(* CoDeSys 2.3 project: cy-159-wg-004.pro *)
(* Title: ClevergyAS - Albino E-02 *)
(* Version: 1.25 *)
(* Author: Andrea Ravasio *)
(* Libraries: mod_com.lib 2.12.10 13:48:32, SerComm.lib 31.5.11 07:54:36, Serial_Interface_01.lib 22.4.13 11:50:14, Standard.lib 2.12.10 13:48:34, Util.lib 26.9.14 09:12:46, Modb_l05.lib 13.5.15 09:30:08, Visual.lib 2.12.10 13:48:34, Ethernet.lib 2.12.10 13:48:32, WagoLibIdent.lib 25.2.13 10:12:16, WagoLibMBX_01.lib 20.3.12 15:32:40, WagoLibStatus.lib 2.12.10 13:48:32, SysLibFile.lib 2.12.10 13:48:34, SysLibRtc.lib 2.12.10 13:48:32, SysLibSockets.lib 10.2.11 08:20:54, SysLibEvent.lib 2.12.10 13:48:34, SysLibPlcCtrl.lib 2.12.10 13:48:32, SysLibCallback.lib 2.12.10 13:48:32, WagoLibModbus_IP_01.lib 24.7.13 14:05:58, WagoLibInfo.lib 25.2.13 09:58:44 *)

(* PLC configuration (modules and I/O channels)
0750-1506 8DI / 8DO 24V DC 0.5A [Type_34_8_Channels] node 0, in %IB128 out %QB120 {INTTypePAAssignment = PLC; INTTypeModule = plugged}
  VPN_ST1 AT %IX64.0 [BOOLOnX_I] Ch_1 Digital input
  LAMP_AL AT %QX60.0 [BOOLOnX_Q] Ch_1 Digital output
  KEY_QE_ST AT %IX64.1 [BOOLOnX_I] Ch_2 Digital input
  AT %QX60.1 [BOOLOnX_Q] Ch_2 Digital output
  AT %IX64.2 [BOOLOnX_I] Ch_3 Digital input
  AT %QX60.2 [BOOLOnX_Q] Ch_3 Digital output
  AT %IX64.3 [BOOLOnX_I] Ch_4 Digital input
  AT %QX60.3 [BOOLOnX_Q] Ch_4 Digital output
  AT %IX64.4 [BOOLOnX_I] Ch_5 Digital input
  AT %QX60.4 [BOOLOnX_Q] Ch_5 Digital output
  AT %IX64.5 [BOOLOnX_I] Ch_6 Digital input
  AT %QX60.5 [BOOLOnX_Q] Ch_6 Digital output
  AT %IX64.6 [BOOLOnX_I] Ch_7 Digital input
  AT %QX60.6 [BOOLOnX_Q] Ch_7 Digital output
  AT %IX64.7 [BOOLOnX_I] Ch_8 Digital input
  AT %QX60.7 [BOOLOnX_Q] Ch_8 Digital output
0750-0652#24 RS-232/RS-485 Interface adjustable (24 Bytes) [Type_30_1_Channels] node 0, in %IB124 out %QB120 {INTTypePAAssignment = PLC; INTTypeModule = plugged}
  AT %IB0 [BYTEOnB_I] First Byte of 24
  AT %QB0 [BYTEOnB_Q] First Byte of 24
0750-0652#24 RS-232/RS-485 Interface adjustable (24 Bytes) [Type_30_1_Channels] node 0, in %IB124 out %QB120 {INTTypePAAssignment = PLC; INTTypeModule = plugged}
  AT %IB24 [BYTEOnB_I] First Byte of 24
  AT %QB24 [BYTEOnB_Q] First Byte of 24
0750-0652#24 RS-232/RS-485 Interface adjustable (24 Bytes) [Type_30_1_Channels] node 0, in %IB148 out %QB144 {INTTypePAAssignment = PLC; INTTypeModule = plugged}
  AT %IB48 [BYTEOnB_I] First Byte of 24
  AT %QB48 [BYTEOnB_Q] First Byte of 24
0750-0652#24 RS-232/RS-485 Interface adjustable (24 Bytes) [Type_30_1_Channels] node 0, in %IB172 out %QB168 {INTTypePAAssignment = PLC; INTTypeModule = plugged}
  AT %IB72 [BYTEOnB_I] First Byte of 24
  AT %QB72 [BYTEOnB_Q] First Byte of 24
0750-0652#24 RS-232/RS-485 Interface adjustable (24 Bytes) [Type_30_1_Channels] node 0, in %IB196 out %QB192 {INTTypePAAssignment = PLC; INTTypeModule = plugged}
  AT %IB96 [BYTEOnB_I] First Byte of 24
  AT %QB96 [BYTEOnB_Q] First Byte of 24
AI_PX01 AT %IW60 [WORDOnW_I] Ch_1 Input word
AI_PX02 AT %IW61 [WORDOnW_I] Ch_2 Input word
AI_PX03 AT %IW62 [WORDOnW_I] Ch_1 Input word
AI_PX04 AT %IW63 [WORDOnW_I] Ch_2 Input word
Fieldbus variables [FB_VARS] node 1, in %IB0 out %QB0
Flag variables [FLAG_VARS] node 2, in %IB0 out %QB0
Modbus-Master [MB_MASTER] node 3, in %IB0 out %QB0
*)

(* Global variable list: Global_Constants *)
VAR_GLOBAL CONSTANT

	Plant_NAME			: STRING :='cySN: 159 cyVER: Supervisione Eredi Gnutti  ';
	Plant_SN			: DWORD  :=159;	(* S/N Impianto di telecontrollo *)
	Plant_SW_VER		: WORD   :=0;	(* Versione SW installata *)


(* Configurazione Analizzatori di rete *)

	Plant_ANZ_INEPRO						: BYTE	 :=5;
	MODBUS_INEPRO_MAX_DEVICE		: BYTE:=Plant_ANZ_INEPRO;
	MODBUS_INEPRO_MAX_REG			: BYTE:=26;

	MODBUS_INEPRO_TIME_OUT			:TIME:=T#500MS;
	ANZ_INEPRO_POLLING_TIME			:TIME:=T#4S;


	(* Filesystem *)
	FilesPath  			: STRING :='S:\';

	(* TCP Logger *)
	Logger_SERVER		: STRING:='';
	Logger_IP			: STRING:='178.33.227.41'; (*'192.168.100.3';*)
	Logger_PORT			: WORD  :=80;
	Logger_GETSTART		: STRING:='GET /cygmsrv/hsgm.ashx?';
	Logger_GETEND		: STRING:='$R$N$R$N';
	Logger_CHECK		: STRING:='True';
	Logger_CRLF			: STRING:='$R$N';
	Logger_DataFile		: STRING:='S:\LOG.DAT';
	Logger_DataFileOld	: STRING:='S:\LOG.BCK';
	Logger_IndexFile	: STRING:='S:\LOG.IDX';
	Logger_ConnRetries	: BYTE:=5;
	Logger_RecoverMsgs	: BYTE:=25;

	(* TCP Remote *)
	Remote_PORT			: WORD  :=10;
	Remote_WELCOME		: STRING:='Connected$R$N';
	Remote_OK			: STRING:='OK$R$N';
	Remote_ERROR		: STRING:='ERROR$R$N';

	(* TCP Sockets *)
	MAX_SEND_TCP_SERVER					 : DWORD:=60000;(*60000*)
	MAX_RECEIVE_TCP_SERVER				 : DWORD:=3000;
	MAX_RECEIVE_TCP_SERVER_SOCKET	 	 : DWORD:=1500;
	MAX_SEND_TCP_CLIENT					 : DWORD:=15000;(*15000*)
	MAX_RECEIVE_TCP_CLIENT				 : DWORD:=1500;
	MAX_RECEIVE_TCP_CLIENT_SOCKET		 : DWORD:=1500;
	MAX_RECEIVE_UDP_SERVER				 : INT  :=1472;
	MAX_RECEIVE_UDP_CLIENT				 : INT  :=1472;
	CONNECT_WATCHDOG_TIME				 : TIME :=t#10s;


	(* VISU COLORS *)
	COLOR_RED 			: DWORD:=16#2020F0;
	COLOR_YELLOW		: DWORD:=16#20F0F0;
	COLOR_GREEN			: DWORD:=16#20F020;
	COLOR_GREEN_OFF 	: DWORD:=16#006000;
	COLOR_LBLUE			: DWORD:=16#F0F080;
	COLOR_LIGHT_GREEN	: DWORD := 16#006000;


END_VAR

(* Global variable list: Global_Retain *)
VAR_GLOBAL RETAIN PERSISTENT
	CAL01_Clima : typ_Clima;
	VRD01_Clima : typ_Clima;
	VRD02_Clima : typ_Clima;
	VRD03_Clima : typ_Clima;
	VRD04_Clima : typ_Clima;

	CTL01_Count : DWORD;

	Mode_Manual : BOOL := FALSE;


	DelayAllarmeTemperaturaNonRaggiunta: INT;
	DeltaInterventoAllarmeTempeaturaNonRaggiuta: INT;
	OffsetSetPointManuale: INT;							(* Offset al Setpoint manuale per comensare lo scambiatore *)
	OffsetSetPointManuale2: INT;						(* Offset al Setpoint manuale per comensare lo scambiatore Aggiuntivo *)
	BitAbilitaBoost: BOOL:=TRUE;						(* Abilitiazione Boost *)
	RifOffsetBoost:INT;									(* Offset al Setpoint della Caldaia per azione di Boost *)

	SogliaMinStartAntigelo: INT;
	SogliaMinStopAntigelo: INT;
	BitAbilitaAntigelo: BOOL:=TRUE;


END_VAR

(* Global variable list: Global_Variables *)
VAR_GLOBAL

	SYS    : typ_SYS;
	Logger : typ_Logger;

	Lamp	:	LAMP_AL_GENERALE;

	T_AMB	:	INT;		(* Environment temperature *)






	(* COMPRESSORI NUOVI COM 01*)
	COMPRESSORE01	:obj_COMPRESSORE_NEW := (ID:=1, Address:=1);
	COMPRESSORE05	:obj_COMPRESSORE_NEW := (ID:=5, Address:=2);

	COMPRESSORE02	:obj_COMPRESSORE_OLD := (ID:=2, Address:=1);
	COMPRESSORE03	:obj_COMPRESSORE_OLD := (ID:=3, Address:=2);
	COMPRESSORE04	:obj_COMPRESSORE_OLD := (ID:=4, Address:=3);

	ESSICATORE01	:obj_ESSICATORE_NEW := (ID:=1, Address:=1);
	ESSICATORE02	:obj_ESSICATORE := (ID:=2, Address:=2);

	FPT01:obj_MisPortata_MB:= (ID:=1, Address:=1);

	(** Communication **)
	(* ModBus TCP *)


(*	MODB06	:	obj_MODBUS_TCP 	:= (ID:=6); *)


	FPT02	:obj_MisPortata_ETH := (ID:=2, IP:='192.168.2.75');		(* misuratori di portata *)
	FPT03	:obj_MisPortata_ETH := (ID:=3, IP:='192.168.2.76');		(* misuratori di portata *)
	FPT04	:obj_MisPortata_ETH := (ID:=4, IP:='192.168.2.77');		(* misuratori di portata *)
	FPT05	:obj_MisPortata_ETH := (ID:=5, IP:='192.168.2.78');		(* misuratori di portata *)
	FPT06	:obj_MisPortata_ETH := (ID:=6, IP:='192.168.2.79');		(* misuratori di portata *)
	FPT07	:obj_MisPortata_ETH := (ID:=7, IP:='192.168.2.80');		(* misuratori di portata *)
	FPT08	:obj_MisPortata_ETH := (ID:=8, IP:='192.168.2.81');		(* misuratori di portata *)
	FPT09	:obj_MisPortata_ETH := (ID:=9, IP:='192.168.2.82');		(* misuratori di portata *)
	FPT10	:obj_MisPortata_ETH := (ID:=10, IP:='192.168.2.83');		(* misuratori di portata *)

	(* ModBus RTU  *)
(*	MODB01	:	obj_MODBUS		:= (ID:=1, COM:=2, BAUDRATE:=BAUD_19200,RS485:=TRUE,MB_timeOut:=t#500ms);   *)					 (* ANZ *)
	MODB02	:	obj_MODBUS	:= (ID:=2, COM:=3, BAUDRATE:=BAUD_9600 ,N_STOPBits:=1,RS485:=TRUE,MB_timeOut:=t#500ms);	(* COMPPRESSORI NUOVI *)
	MODB03	:	obj_MODBUS		:= (ID:=3, COM:=4, BAUDRATE:=BAUD_9600,N_STOPBits:=1,RS485:=TRUE,MB_timeOut:=t#500ms);	(* COMPRESSORI VECCHI *)
	MODB04	:	obj_MODBUS_Free		:= (ID:=4, COM:=5, BAUDRATE:=BAUD_9600,N_STOPBits:=1,RS485:=TRUE,MB_timeOut:=t#1s);  (*ESSICATORI *)
	MODB05	:	obj_MODBUS 		:= (ID:=5, COM:=6, BAUDRATE:=BAUD_9600,N_STOPBits:=1,RS485:=TRUE,MB_timeOut:=t#1s);  (*FTP01 *)





	(* Define the handler for the ModBus communication	*)
	MODB01		:	obj_MODBUS_ANZ := (ID:=1, COM:=2,
						(* TIME_OUT_TIME:= TIME_OUT_TIME:=MODBUS_INEPRO_TIME_OUT,*)
						 BAUDRATE:=BAUD_9600,
						  RS485:=TRUE,PARITY:=PARITY_EVEN,STOP_BITS:=STOPBITS_1 );


	ANZ_MODBUS_CONNECTOR_INEPRO	:	ARRAY[1..Plant_ANZ_INEPRO] OF obj_MODBUS_GENERIC_CONNECTOR;
	ANZ_INEPRO									:	ARRAY[1..Plant_ANZ_INEPRO] OF obj_ANZ_INEPRO_PRO380;

	MODBUS_INEPRO_RegDescr 				: ARRAY[1..MODBUS_INEPRO_MAX_DEVICE, 1..MODBUS_INEPRO_MAX_REG] OF STRING(20);
	MODBUS_INEPRO_RegAddress			 : ARRAY[1..MODBUS_INEPRO_MAX_DEVICE, 1..MODBUS_INEPRO_MAX_REG] OF WORD;
	MODBUS_INEPRO_RegQuantity 			: ARRAY[1..MODBUS_INEPRO_MAX_DEVICE, 1..MODBUS_INEPRO_MAX_REG] OF BYTE;
	MODBUS_INEPRO_RegValueType			 : ARRAY[1..MODBUS_INEPRO_MAX_DEVICE, 1..MODBUS_INEPRO_MAX_REG] OF en_Modbus_Reg_Type;




(* CONFIGURAZIONE INGRESSI ANALOGICI 4-20mA  *)

	PX01  : obj_AI_GEN	:= ( ID:=1 ,
								SogliaHL:=4096 ,   	 	(* Soglia Sonda Aperta = 2,5mA *)
								SogliaHH:=32767,	 	(* Soglia Sonda CC = 20mA *)
								SogliaWL:=10, 			(* Soglia WRN Bassa  *)
								SogliaWH:=140,			(* Soglia WRN Alta   *)
								PuntoMinX:=0, 		   	 (* Scalatura Minima vedi data di targa sonda 0 bar *)
								PuntoMaxX:=160,			(* Scalatura Massima Vedi data di targa Sonda 16.0bar *)
								PuntoMinY:=6553,			(* Valore minimio per scalatura = 4mA *)
								PuntoMaxY:=32767,		(* Valore Massimo per Scalatura = 20mA *)
								Decimali:=0,				(* Decimali da ottenere durante la scalatura *)
								TipoSensore:='PPV'		(* Riferimento nle file LOG *)
								);

	PX02  : obj_AI_GEN	:= ( ID:=2 ,
								SogliaHL:=4096 ,   	 	(* Soglia Sonda Aperta = 2,5mA *)
								SogliaHH:=32767,	 	(* Soglia Sonda CC = 20mA *)
								SogliaWL:=10, 			(* Soglia WRN Bassa *)
								SogliaWH:=120,			(* Soglia WRN Alta *)
								PuntoMinX:=0, 		   	 (* Scalatura Minima vedi data di targa sonda  0 bar*)
								PuntoMaxX:=160,			(* Scalatura Massima Vedi data di targa Sonda 16.0bar  *)
								PuntoMinY:=6553,			(* Valore minimio per scalatura = 4mA *)
								PuntoMaxY:=32767,		(* Valore Massimo per Scalatura = 20mA *)
								Decimali:=0,				(* Decimali da ottenere durante la scalatura *)
								TipoSensore:='PPV'		(* Riferimento nle file LOG *)
								);

	PX03  : obj_AI_GEN	:= ( ID:=3 ,
								SogliaHL:=4096 ,   	 	(* Soglia Sonda Aperta = 2,5mA *)
								SogliaHH:=32767,	 	(* Soglia Sonda CC = 20mA *)
								SogliaWL:=10, 			(* Soglia WRN Bassa  = *)
								SogliaWH:=120,			(* Soglia WRN Alta  =  *)
								PuntoMinX:=0, 		   	 (* Scalatura Minima vedi data di targa sonda  0 bar*)
								PuntoMaxX:=160,			(* Scalatura Massima Vedi data di targa Sonda 16.0bar *)
								PuntoMinY:=6553,			(* Valore minimio per scalatura = 4mA *)
								PuntoMaxY:=32767,		(* Valore Massimo per Scalatura = 20mA *)
								Decimali:=0,				(* Decimali da ottenere durante la scalatura *)
								TipoSensore:='PPV'		(* Riferimento nle file LOG *)
								);

	PX04  : obj_AI_GEN	:= ( ID:=4 ,
								SogliaHL:=4096 ,   	 	(* Soglia Sonda Aperta = 2,5mA *)
								SogliaHH:=32767,	 	(* Soglia Sonda CC = 20mA *)
								SogliaWL:=10, 			(* Soglia WRN Bassa  =  *)
								SogliaWH:=120,			(* Soglia WRN Alta  =  *)
								PuntoMinX:=0, 		   	 (* Scalatura Minima vedi data di targa sonda 0 bar *)
								PuntoMaxX:=160,			(* Scalatura Massima Vedi data di targa Sonda 16.0bar *)
								PuntoMinY:=6553,			(* Valore minimio per scalatura = 4mA *)
								PuntoMaxY:=32767,		(* Valore Massimo per Scalatura = 20mA *)
								Decimali:=0,				(* Decimali da ottenere durante la scalatura *)
								TipoSensore:='PPV'		(* Riferimento nle file LOG *)
								);





(* interblocchi comunicazione modbus *)

	NodoDaInterrogareCompressoreNuovo: BYTE;
	InibiscoModbusCompressoreNuovo: BOOL;

	NodoDaInterrogareCompressoreVecchio: BYTE;
	InibiscoModbusCompressoreVecchio: BOOL;

	NodoDaInterrogareMisuratoreDiPortata: BYTE;
	InibiscoModbusMisuratoreDiPortata: BOOL;

	NodoDaInterrogareMisuratoreDiPortata_ETH: BYTE;

	NodoDaInterrogareEssicatore: BYTE;
	InibiscoModbusEssicatore: BOOL;



END_VAR

(* Data type in LON/Enumerations *)
TYPE alarm_type_t :
(
	AL_HEADER := -13,
	AL_FOOTER := -12,
	AL_DEBUG := -11,
	AL_INFO := -10,
	AL_SYSTEM_INFO := -6,
	AL_VALUE_INVALID := -5,
	AL_CONSTANT := -4,
	AL_OFFLINE := -3,
	AL_UNKNOWN := -2,
	AL_NUL := -1,
	AL_NO_CONDITION := 0,
	AL_ALM_CONDITION := 1,
	AL_TOT_SVC_ALM_1 := 2,
	AL_TOT_SVC_ALM_2 := 3,
	AL_TOT_SVC_ALM_3 := 4,
	AL_LOW_LMT_CLR_1 := 5,
	AL_LOW_LMT_CLR_2 := 6,
	AL_HIGH_LMT_CLR_1 := 7,
	AL_HIGH_LMT_CLR_2 := 8,
	AL_LOW_LMT_ALM_1 := 9,
	AL_LOW_LMT_ALM_2 := 10,
	AL_HIGH_LMT_ALM_1 := 11,
	AL_HIGH_LMT_ALM_2 := 12,
	AL_FIR_ALM := 13,
	AL_FIR_PRE_ALM := 14,
	AL_FIR_TRBL := 15,
	AL_FIR_SUPV := 16,
	AL_FIR_TEST_ALM := 17,
	AL_FIR_TEST_PRE_ALM := 18,
	AL_FIR_ENVCOMP_MAX := 19,
	AL_FIR_MONITOR_COND := 20,
	AL_FIR_MAINT_ALERT := 21,
	AL_FATAL_ERROR := 30,
	AL_ERROR := 31,
	AL_WARNING := 32
);
END_TYPE

(* Data type in DT_ANZ *)
TYPE en_ANZ_Type :
(
	THREE_PHASE			:=0,
	MONO_PHASE			:=1
);
END_TYPE

(* Data type in Errors *)
TYPE en_Logger_ErrLev :
(
	EL_Log			:=0,
	EL_Wrn			:=1,
	EL_Alarm		:=2,
	EL_AlarmStop	:=3
);
END_TYPE

(* Data type in Errors *)
TYPE en_Logger_Status :
(
	S_Logger_UNKNOWN := 0,
	S_Logger_IDLE,
	S_Logger_WAITCONN,
	S_Logger_WAITTX,
	S_Logger_WAITRESP,
	S_Logger_ERROR
);
END_TYPE

(* Data type *)
TYPE en_Modbus_Reg_Type :
(
	VALUE_REAL		:=0,
	VALUE_LONG		:=4
);
END_TYPE

(* Data type *)
TYPE en_SYS_Objects :
(
	EO_SYS		:=0,  (* PLC *)
	EO_VPN		:=1,  (* VPN *)
	EO_DOOR		:=2,  (* Door & access control *)

	EO_CAL		:=10, (* Caldaia *)
	EO_CIR		:=11, (* Circolatore *)
	EO_CRON		:=12, (* Crono-termostato *)
	EO_VRD		:=13, (* Valvola miscelatore pannelli *)
	EO_CTL		:=14, (* Contalitri *)
	EO_CTB		:=15, (* Contabilizzatore *)
	EO_TPV		:=16, (* Temperature probes values *)
	EO_PPV		:=17, (* Pressure probes values *)
	EO_PBV		:=18, (* Over-Pressure Alarms *)
	EO_TBV		:=19, (* Over-Temperature Alarms *)
	EO_PMV		:=20, (* Under-Pressure Alarms *)
	EO_GRU		:=21, (* Gruppo termico *)
	EO_PDC		:=22, (* Pompa di calore *)
	EO_SOL		:=23, (* Pannello solare termico *)
	EO_ESOL		:=24, (* Pannello solare fotovoltaico *)
	EO_GAS		:=25, (* Contatore GAS *)
	EO_PORT		:=26, (* Misuratore di portata *)
	EO_FPV		:=27, (* Flow probes values *)
	EO_ANZ		:=28, (* Analizzatore di rete *)
	EO_SCA		:=29, (* Signal Control Alarms *)
	EO_LUX		:=30, (* Base Illumination point *)
	EO_LUXM		:=31, (* Metered Illumination point *)
	EO_PSG		:=32, (* Sensore di passaggio *)
	EO_HVAC		:=33, (* Heating, Ventilating and Air Conditioning *)
	EO_HYGRV	:=34, (* Relative Humidity sensors value *)
	EO_COOV		:=35, (* Carbon Dioxide CO2 sensors value *)
	EO_INV		:=36, (* Inverter *)
	EO_STR		:=37, (* Smart string box *)

	EO_CIRD		:=39, (* Double CIR *)
	EO_ACS		:=40, (* Hot domestic water *)
	EO_FRG		:=41, (* Frigo *)
	EO_THER		:=42, (* Thermostat *)
	EO_CIRM		:=43, (* Modbus CIR *)
	EO_CIRDM	:=44, (* Modbus double CIR *)
	EO_UTA		:=47, (* Modbus double CIR *)

	EO_FPT		:=53, (* Flow Pressure Temperature	FPTxx *)


	EO_ZGW			:=200,  (* ZigBee - Gateway *)
	EO_ZRM			:=201,	(* ZigBee - Repeater *)
	EO_ZREL			:=202,	(* ZigBee - Actuator rele *)
	EO_ZTHL			:=203,	(* ZigBee - Temperature Sensor *)

	EO_ASGW			:=250,	(* ASi - Gateway *)
	EO_ASCBI		:=251,	(* ASi - Input Board, Ciabatta *)

	EO_LON			:=1000, (* Bus - LON *)
	EO_MODBUS		:=1001, (* Bus - MODBUS *)
	EO_MBUS			:=1002, (* Bus - M-BUS *)
	EO_MODBUS_TCP	:=1003, (* Bus - MODBUS TCP *)




	EO_COMPINGRR		:=10000,		(*Compressore Ingerson Rand R225 NE *)
	EO_COMPINGRML	:=	10001,		(*Compressore Ingerson Rand ML250SSR *)
	EO_ESC				:=	10002,		(*Essicatore *)





	EO_GENERIC		:=9000, (* Generic dataset *)
	EO_EXPO			:=9001 (* EXPO dataset *)
);
END_TYPE

(* Data type *)
TYPE en_SYS_Status :
(
	S_UNKNOWN  := 0,
	S_STARTUP,
	S_INIT_RTC,
	S_INIT_VAR,
	S_AUTOTEST,
	S_RUNNING,
	S_SHUTDOWN,
	S_HALT
);
END_TYPE

(* Data type in LON/Enumerations *)
TYPE file_request_t :
(
	FR_NUL := -1,
	FR_OPEN_TO_SEND := 0,
	FR_OPEN_TO_RECEIVE := 1,
	FR_CLOSE_FILE := 2,
	FR_CLOSE_DELETE_FILE := 3,
	FR_DIRECTORY_LOOKUP := 4,
	FR_OPEN_TO_SEND_RA := 5,
	FR_OPEN_TO_RECEIVE_RA := 6
);
END_TYPE

(* Data type in LON/Enumerations *)
TYPE file_status_t :
(
	FS_NUL := -1,
	FS_XFER_OK := 0,
	FS_LOOKUP_OK := 1,
	FS_OPEN_FAIL := 2,
	FS_LOOKUP_ERR := 3,
	FS_XFER_UNDERWAY := 4,
	FS_IO_ERR := 5,
	FS_TIMEOUT_ERR := 6,
	FS_WINDOW_ERR := 7,
	FS_AUTH_ERR := 8,
	FS_ACCESS_UNAVAIL := 9,
	FS_SEEK_INVALID := 10,
	FS_SEEK_WAIT := 11
);
END_TYPE

(* Data type in LON/Enumerations *)
TYPE hvac_t :
(
	HVAC_NUL := -1,
	HVAC_AUTO := 0,
	HVAC_HEAT := 1,
	HVAC_MRNG_WRMUP := 2,
	HVAC_COOL := 3,
	HVAC_NIGHT_PURGE := 4,
	HVAC_PRE_COOL := 5,
	HVAC_OFF := 6,
	HVAC_TEST := 7,
	HVAC_EMERG_HEAT := 8,
	HVAC_FAN_ONLY := 9,
	HVAC_FREE_COOL := 10,
	HVAC_ICE := 11,
	HVAC_MAX_HEAT := 12,
	HVAC_ECONOMY := 13,
	HVAC_DEHUMID := 14,
	HVAC_CALIBRATE := 15,
	HVAC_EMERG_COOL := 16,
	HVAC_EMERG_STEAM := 17,
	HVAC_MAX_COOL := 18,
	HVAC_HVC_LOAD := 19,
	HVAC_NO_LOAD := 20
);
END_TYPE

(* Data type in LON/Enumerations *)
TYPE object_request_t :
(
	RQ_NUL := -1,
	RQ_NORMAL := 0,
	RQ_DISABLED := 1,
	RQ_UPDATE_STATUS := 2,
	RQ_SELF_TEST := 3,
	RQ_UPDATE_ALARM := 4,
	RQ_REPORT_MASK := 5,
	RQ_OVERRIDE := 6,
	RQ_ENABLE := 7,
	RQ_RMV_OVERRIDE := 8,
	RQ_CLEAR_STATUS := 9,
	RQ_CLEAR_ALARM := 10,
	RQ_ALARM_NOTIFY_ENABLED := 11,
	RQ_ALARM_NOTIFY_DISABLED := 12,
	RQ_MANUAL_CTRL := 13,
	RQ_REMOTE_CTRL := 14,
	RQ_PROGRAM := 15,
	RQ_CLEAR_RESET := 16,
	RQ_RESET := 17,
	RQ_CLEAR_LOG := 18,
	RQ_LOAD_PROGRAM := 19,
	RQ_RUN_PROGRAM := 20,
	RQ_HALT_PROGRAM := 21,
	RQ_RESTART_PROGRAM := 22,
	RQ_UNLOAD_PROGRAM := 23,
	RQ_STEP_PROGRAM := 24
);
END_TYPE

(* Data type in LON/Enumerations *)
TYPE priority_level_t :
(
	PR_NUL := -1,
	PR_LEVEL_0 := 0,
	PR_LEVEL_1 := 1,
	PR_LEVEL_2 := 2,
	PR_LEVEL_3 := 3,
	PR_1 := 4,
	PR_2 := 5,
	PR_3 := 6,
	PR_4 := 7,
	PR_6 := 8,
	PR_8 := 9,
	PR_10 := 10,
	PR_16 := 11
);
END_TYPE

(* Data type in DT_ANZ *)
(*
	typ_ANZ_3P 

	Data that each ANZ 3-phase block must provide (to the Clevergy platform).
*)
TYPE typ_ANZ :
STRUCT

	(* voltages *)
	V_L1N		:	DWORD;	(* V *)
	V_L2N		:	DWORD;
	V_L3N		:	DWORD;
	V_L1L2		:	DWORD;
	V_L2L3		:	DWORD;
	V_L3L1		:	DWORD;

	(* frequency *)
	FREQ		:	DWORD;	(* E-3 Hz *) (* rif. L1 *)

	(* currents *)
	I_L1			:	DWORD;	(* E-3 A *)
	I_L2			:	DWORD;
	I_L3			:	DWORD;
	I_L1_Max		:	DWORD;	(* E-3 A *)
	I_L2_Max		:	DWORD;
	I_L3_Max		:	DWORD;

	(* power factors *)
	PF_L1		:	DINT;	(* E-3 *)
	PF_L2		:	DINT;
	PF_L3		:	DINT;

	(* active powers *)
	P_3P			:	DINT;   (* W *)
	P_3P_Avg		:	DINT;
	P_3P_Max	:	DINT:=0;

	(* reactive powers *)
	Q_3P		:	DINT;	(* VAr *)
	Q_3P_Max	:	DINT:=-2147483648;	(* VAr *)

	(* active energy *)
	WH_3P		:	DWORD;	(* Wh *)

	(* reactive energy *)
	VARH_3P		:	DINT;	(* VArh *)

	(* cosphi *)
	COSPHI_L1		:	DINT;	(* E-3 *)
	COSPHI_L2		:	DINT;	(* E-3 *)
	COSPHI_L3		:	DINT;	(* E-3 *)

END_STRUCT
END_TYPE

(* Data type in DT_ANZ_INEPRO_PRO380 *)
TYPE typ_ANZ_INEPRO_PRO380 :
STRUCT

		rTotalActivePower					: REAL;
		rTotalReactivePower				: REAL;
		rTotalApparentPower				: REAL;
		rTotalPowerFactorPF				: REAL;
		rTotalActiveEnergy					: REAL;
		rTotalReactiveEnergy				: REAL;

		arCurrent							: ARRAY[1..3] OF REAL;
		arVoltage_L_N						: ARRAY[1..3] OF REAL;
		arActivePower						: ARRAY[1..3] OF REAL;
		arReactivePower					: ARRAY[1..3] OF REAL;
		arApparentPower					: ARRAY[1..3] OF REAL;

		arPowerFactorPF					: ARRAY[1..3] OF REAL;
		arFrequency						:REAL;


		rMaximumCurrentL1			: REAL;
		rMaximumCurrentL2				: REAL;
		rMaximumCurrentL3			: REAL;


		rMaximumTotalActivePower			: REAL :=0;
		rAverageTotalActivePower 			: REAL :=0;

		rMaximumTotalReactivePower		: REAL :=0;

END_STRUCT
END_TYPE

(* Data type in DT_ANZ *)
(*
	typ_ANZ_3P 

	Data that each ANZ 3-phase block must provide (to the Clevergy platform).
*)
TYPE typ_ANZ_REAL :
STRUCT

	(* voltages *)
	V_L1N		:	REAL;	(* V *)
	V_L2N		:	REAL;
	V_L3N		:	REAL;
	V_L1L2		:	REAL;
	V_L2L3		:	REAL;
	V_L3L1		:	REAL;

	(* frequency *)
	FREQ		:	REAL;	(* E-3 Hz *) (* rif. L1 *)

	(* currents *)
	I_L1			:	REAL;	(* E-3 A *)
	I_L2			:	REAL;
	I_L3			:	REAL;
	I_L1_Max		:	REAL;	(* E-3 A *)
	I_L2_Max		:	REAL;
	I_L3_Max		:	REAL;

	(* power factors *)
	PF_L1		:	REAL;	(* E-3 *)
	PF_L2		:	REAL;
	PF_L3		:	REAL;

	(* active powers *)
	P_3P			:	REAL;   (* W *)
	P_3P_Avg		:	REAL;
	P_3P_Max	:	REAL:=0;

	(* reactive powers *)
	Q_3P		:	REAL;	(* VAr *)
	Q_3P_Max	:	REAL:=-2147483648;	(* VAr *)

	(* active energy *)
	WH_3P		:	REAL;	(* Wh *)

	(* reactive energy *)
	VARH_3P		:	REAL;	(* VArh *)

	(* cosphi *)
	COSPHI_L1		:	REAL;	(* E-3 *)
	COSPHI_L2		:	REAL;	(* E-3 *)
	COSPHI_L3		:	REAL;	(* E-3 *)

END_STRUCT
END_TYPE

(* Data type in Plant_Objects *)
TYPE typ_Clima : (* CURVA CLIMATICA *)
STRUCT
	InitOK:		BOOL;
	Points: 	ARRAY [0..10] OF POINT;
END_STRUCT
END_TYPE

(* Data type in Plant_Objects *)
TYPE typ_Cron_Calendar :
STRUCT
	Profile		: ARRAY[0..384] OF BYTE;
END_STRUCT
END_TYPE

(* Data type in Plant_Objects *)
TYPE typ_Cron_Jolly :
STRUCT
	Start		: DT;
	End			: DT;
	Temp		: WORD;
	Flags		: WORD; (* B0:Enabled B1..B15:Unused *)
END_STRUCT
END_TYPE

(* Data type in Plant_Objects *)
TYPE typ_Cron_Profile :
STRUCT
	Flags		: WORD;
	Setpoint	: ARRAY [0..95] OF WORD;
END_STRUCT
END_TYPE

(* Data type in Errors *)
TYPE typ_Logger :
STRUCT
	Status		: en_Logger_Status;

	SendReq		: BOOL;
	SendIdx		: DWORD;
	SendData	: ARRAY [0..MAX_SEND_TCP_CLIENT] OF BYTE;
	SendLen		: DINT;

	TData		: ARRAY [0..MAX_SEND_TCP_CLIENT] OF BYTE;
	TLen		: DINT;

	LastIdxPos	: DWORD;

	(* Temporary variables used by objects *)
	s1			: STRING(256);
	i1			: WORD;


END_STRUCT
END_TYPE

(* Data type in Plant_Objects *)
TYPE typ_MODBUS_VAR : (* Gestione parametri MODBUS *)
STRUCT
	SlaveAddress	: BYTE;
	FunCode			: BYTE;
	FunAddress		: WORD;
	Refresh_Time	: BYTE; (* 0:No refresh x:Refresh in seconds *)
	Refresh_Cnt		: BYTE; (* INTERNAL *)
	Variable		: POINTER TO WORD;
	Variable_Size	: BYTE;
	Variable_Mirror : WORD; (* INTERNAL [Force refresh on read variables when <>0] *)
END_STRUCT
END_TYPE

(* Data type in Plant_Objects *)
TYPE typ_MODBUS_VAR_ANZ : (* Gestione parametri MODBUS *)
STRUCT
	SlaveAddress	: BYTE;
	FunCode			: BYTE;
	FunAddress		: WORD;
	Refresh_Time	: BYTE; (* 0:No refresh x:Refresh in seconds *)
	Refresh_Cnt		: BYTE; (* INTERNAL *)
	Variable		: POINTER TO ARRAY [0..124] OF WORD;	(* For classical ModBus it has to be equal to "typModbusResponse.Data"
																that is an array of 125 word ([0..124]) *)
	Variable_Size	: BYTE;
	Variable_Mirror : WORD; (* INTERNAL [Force refresh on read variables when <>0] *)
END_STRUCT
END_TYPE

(* Data type *)
TYPE typ_SYS :
STRUCT
	Status			: en_SYS_Status;
	Warning			: BOOL;
	Alarm			: BOOL;
	AlarmStop		: BOOL;

	Time_LogString	: STRING;
	Time_Year		: WORD;
	Time_Month		: BYTE;
	Time_Day		: BYTE;

	Time_CT_DT		: DT;
	Time_CT_Day		: WORD;
	Time_CT_Quarter	: BYTE;

	LastLogs_Idx	: BYTE;
	LastLogs_Dat	: ARRAY[0..5] OF STRING;
	LastLogs_Msg	: ARRAY[0..5] OF STRING;

END_STRUCT
END_TYPE

(* Data type in LON/NetworkVariables *)
TYPE typSnvtAlarm : 
STRUCT
	abLocation : ARRAY[0..5] OF BYTE;
	wObjectId : WORD;
	bAlarmType : BYTE (* enum type alarm_type_t *);
	bPriorityLevel : BYTE (* enum type priority_level_t *);
	wIndexToSnvt : WORD;
	abValue : ARRAY[0..3] OF BYTE;
	wYear : WORD;
	bMonth : BYTE;
	bDay : BYTE;
	bHour : BYTE;
	bMinute : BYTE;
	bSecond : BYTE;
	wMillisecond : WORD;
	abAlarmLimit : ARRAY[0..3] OF BYTE;
	bStatusInformation : BYTE; (* bit allocation of bStatusInformation:
	bit 0: NVI update counter LSB
	bit 1: NVI update counter
	bit 2: NVI update counter
	bit 3: NVI update counter MSB
	bit 4: timeout for NVI occurs (MaxRcvTime expired)
	bit 5: reserved
	bit 6: reserved
	bit 7: force NVO update *)
	bInternalUseOnly : BYTE; (* Do not use this byte in your application! *)
END_STRUCT
END_TYPE

(* Data type in LON/NetworkVariables *)
TYPE typSnvtFilePos : 
STRUCT
	diRwPtr : DINT;
	wRwLength : WORD;
	bStatusInformation : BYTE; (* bit allocation of bStatusInformation:
	bit 0: NVI update counter LSB
	bit 1: NVI update counter
	bit 2: NVI update counter
	bit 3: NVI update counter MSB
	bit 4: timeout for NVI occurs (MaxRcvTime expired)
	bit 5: reserved
	bit 6: reserved
	bit 7: force NVO update *)
	bInternalUseOnly : BYTE; (* Do not use this byte in your application! *)
END_STRUCT
END_TYPE

(* Data type in LON/NetworkVariables *)
TYPE typSnvtFileReq : 
STRUCT
	bRequest : BYTE (* enum type file_request_t *);
	wIndex : WORD;
	wReceiveTimeout : WORD;
	abDestAddress : ARRAY[0..4] OF BYTE (* union declaration *);
	bAuthOn : BYTE;
	bPrioOn : BYTE;
	bStatusInformation : BYTE; (* bit allocation of bStatusInformation:
	bit 0: NVI update counter LSB
	bit 1: NVI update counter
	bit 2: NVI update counter
	bit 3: NVI update counter MSB
	bit 4: timeout for NVI occurs (MaxRcvTime expired)
	bit 5: reserved
	bit 6: reserved
	bit 7: force NVO update *)
	bInternalUseOnly : BYTE; (* Do not use this byte in your application! *)
END_STRUCT
END_TYPE

(* Data type in LON/NetworkVariables *)
TYPE typSnvtFileStatus : 
STRUCT
	bStatus : BYTE (* enum type file_status_t *);
	wNumberOfFiles : WORD;
	wSelectedFile : WORD;
	abAdr : ARRAY[0..21] OF BYTE (* union declaration *);
	bStatusInformation : BYTE; (* bit allocation of bStatusInformation:
	bit 0: NVI update counter LSB
	bit 1: NVI update counter
	bit 2: NVI update counter
	bit 3: NVI update counter MSB
	bit 4: timeout for NVI occurs (MaxRcvTime expired)
	bit 5: reserved
	bit 6: reserved
	bit 7: force NVO update *)
	bInternalUseOnly : BYTE; (* Do not use this byte in your application! *)
END_STRUCT
END_TYPE

(* Data type in LON/NetworkVariables *)
TYPE typSnvtHvacMode : 
STRUCT
	bSnvtHvacMode : BYTE (* enum type hvac_t *);
	bStatusInformation : BYTE; (* bit allocation of bStatusInformation:
	bit 0: NVI update counter LSB
	bit 1: NVI update counter
	bit 2: NVI update counter
	bit 3: NVI update counter MSB
	bit 4: timeout for NVI occurs (MaxRcvTime expired)
	bit 5: reserved
	bit 6: reserved
	bit 7: force NVO update *)
	bInternalUseOnly : BYTE; (* Do not use this byte in your application! *)
END_STRUCT
END_TYPE

(* Data type in LON/NetworkVariables *)
TYPE typSnvtObjRequest : 
STRUCT
	wObjectId : WORD;
	bObjectRequest : BYTE (* enum type object_request_t *);
	bStatusInformation : BYTE; (* bit allocation of bStatusInformation:
	bit 0: NVI update counter LSB
	bit 1: NVI update counter
	bit 2: NVI update counter
	bit 3: NVI update counter MSB
	bit 4: timeout for NVI occurs (MaxRcvTime expired)
	bit 5: reserved
	bit 6: reserved
	bit 7: force NVO update *)
	bInternalUseOnly : BYTE; (* Do not use this byte in your application! *)
END_STRUCT
END_TYPE

(* Data type in LON/NetworkVariables *)
TYPE typSnvtObjStatus : 
STRUCT
	wObjectId : WORD;
	bBitfieldByteOffset2 : BYTE (* bit field *);
	bBitfieldByteOffset3 : BYTE (* bit field *);
	bBitfieldByteOffset4 : BYTE (* bit field *);
	bBitfieldByteOffset5 : BYTE (* bit field *);
	bStatusInformation : BYTE; (* bit allocation of bStatusInformation:
	bit 0: NVI update counter LSB
	bit 1: NVI update counter
	bit 2: NVI update counter
	bit 3: NVI update counter MSB
	bit 4: timeout for NVI occurs (MaxRcvTime expired)
	bit 5: reserved
	bit 6: reserved
	bit 7: force NVO update *)
	bInternalUseOnly : BYTE; (* Do not use this byte in your application! *)
END_STRUCT
END_TYPE

(* Data type in LON/NetworkVariables *)
TYPE typSnvtState : 
STRUCT
	bBitfieldByteOffset0 : BYTE (* bit field *);
	bBitfieldByteOffset1 : BYTE (* bit field *);
	bStatusInformation : BYTE; (* bit allocation of bStatusInformation:
	bit 0: NVI update counter LSB
	bit 1: NVI update counter
	bit 2: NVI update counter
	bit 3: NVI update counter MSB
	bit 4: timeout for NVI occurs (MaxRcvTime expired)
	bit 5: reserved
	bit 6: reserved
	bit 7: force NVO update *)
	bInternalUseOnly : BYTE; (* Do not use this byte in your application! *)
END_STRUCT
END_TYPE

(* Data type in LON/NetworkVariables *)
TYPE typSnvtSwitch : 
STRUCT
	bValue : BYTE;
	siState : SINT;
	bStatusInformation : BYTE; (* bit allocation of bStatusInformation:
	bit 0: NVI update counter LSB
	bit 1: NVI update counter
	bit 2: NVI update counter
	bit 3: NVI update counter MSB
	bit 4: timeout for NVI occurs (MaxRcvTime expired)
	bit 5: reserved
	bit 6: reserved
	bit 7: force NVO update *)
	bInternalUseOnly : BYTE; (* Do not use this byte in your application! *)
END_STRUCT
END_TYPE

(* Data type in LON/NetworkVariables *)
TYPE typSnvtTempP :
STRUCT
	iSnvtTempP : INT;
	bStatusInformation : BYTE; (* bit allocation of bStatusInformation:
	bit 0: NVI update counter LSB
	bit 1: NVI update counter
	bit 2: NVI update counter
	bit 3: NVI update counter MSB
	bit 4: timeout for NVI occurs (MaxRcvTime expired)
	bit 5: reserved
	bit 6: reserved
	bit 7: force NVO update *)
	bInternalUseOnly : BYTE; (* Do not use this byte in your application! *)
END_STRUCT
END_TYPE

(* Data type in LON/NetworkVariables *)
TYPE typSnvtTimeStamp : 
STRUCT
	iYear : INT;
	bMonth : BYTE;
	bDay : BYTE;
	bHour : BYTE;
	bMinute : BYTE;
	bSecond : BYTE;
	bStatusInformation : BYTE; (* bit allocation of bStatusInformation:
	bit 0: NVI update counter LSB
	bit 1: NVI update counter
	bit 2: NVI update counter
	bit 3: NVI update counter MSB
	bit 4: timeout for NVI occurs (MaxRcvTime expired)
	bit 5: reserved
	bit 6: reserved
	bit 7: force NVO update *)
	bInternalUseOnly : BYTE; (* Do not use this byte in your application! *)
END_STRUCT
END_TYPE

(* POU PLC_PRG, ST *)
PROGRAM PLC_PRG
VAR
	Timer1: TON; (* Fast controls tick *)
	Timer2: TON; (* Plant control tick *)
	Timer3: TON; (* Logger timer *)


	status : BYTE;
	i	  : BYTE;



	HMI_AggiornaLog: BOOL;

	TempoCilcoETH: TON;
	StepETH: INT;


	Timer4: TON;
	IndiceArraRet: INT;
	pippo: BOOL;
	k: INT;
	CreaFile: obj_CreaFile;
	arra: BOOL;
	ArrayDaSalvare: ARRAY [1..80,0..60] OF STRING(10);
	record: INT;
	x: INT;


	EseguiLog: INT;
	Ton_pausaTrig: TON;
	R_TrigAggiornaLog: R_TRIG;


	TempoLog: TIME := t#500ms;
END_VAR

VAR RETAIN

END_VAR


VAR_INPUT
	RichiestaDaRemoto:BOOL;

END_VAR
(******************************************************************************
 ****                           MAIN TASK CODE                             ****
 ******************************************************************************

	Network setup:
		IP  = 192.168.2.73 | MSK = 255.255.255.0
		GW	= 192.168.2.254 | DNS = 192.168.100.1
		SNTP = 193.204.114.232 (3600s) ==> 192.168.100.3
*)





(*==============================*)
(*===== Main status machine ====*)
(*==============================*)


Main_Stm();

(*==============================*)
(*== Running cycle operations ==*)
(*==============================*)

IF SYS.Status>S_INIT_VAR THEN




	(* ModBus *)
	MODB02();

	COMPRESSORE01(ModBus:=MODB02);
	COMPRESSORE05(ModBus:=MODB02);

	NodoDaInterrogareCompressoreNuovo:=LIMIT(1,NodoDaInterrogareCompressoreNuovo,3);
	IF NodoDaInterrogareCompressoreNuovo>2 THEN NodoDaInterrogareCompressoreNuovo:=1;END_IF;


	(* ModBus *)
	MODB03();

	COMPRESSORE02(ModBus:=MODB03);
	COMPRESSORE03(ModBus:=MODB03);
	COMPRESSORE04(ModBus:=MODB03);

	NodoDaInterrogareCompressoreVecchio:=LIMIT(1,NodoDaInterrogareCompressoreVecchio,4);
	IF NodoDaInterrogareCompressoreVecchio>3 THEN NodoDaInterrogareCompressoreVecchio:=1;END_IF;


	(* ModBus *)
	MODB04();


(*	ESSICATORE01(ModBus:=MODB04); *)
	ESSICATORE02(ModBus:=MODB04);

	NodoDaInterrogareEssicatore:=LIMIT(1,NodoDaInterrogareEssicatore,3);
	IF NodoDaInterrogareEssicatore>2 THEN NodoDaInterrogareEssicatore:=2;END_IF;  (**** ma modificare nel caso si inserisca anche il nodo 1 ***)





	(* ModBus *)
	MODB05();

	FPT01(ModBus:=MODB05);

	NodoDaInterrogareMisuratoreDiPortata:=LIMIT(1,NodoDaInterrogareMisuratoreDiPortata,2);
	IF NodoDaInterrogareMisuratoreDiPortata>1 THEN NodoDaInterrogareMisuratoreDiPortata:=1;END_IF;





	TempoCilcoETH(IN:= NOT TempoCilcoETH.Q , PT:=t#1s , Q=> , ET=> );
	IF TempoCilcoETH.Q THEN StepETH:=StepETH+1;END_IF


 	FPT02();
	FPT03();
	FPT04();
	FPT05();
	FPT06();
	FPT07();
	FPT08();
	FPT09();
	FPT10();



	(*MODB06(); *)

	(* FPT02(startCom:=StepETH=2,MODBUS:=MODB06); *)
	(* FPT03(startCom:=StepETH=3  ,MODBUS:=MODB06);
	 FPT04(startCom:=StepETH=4 ,MODBUS:=MODB06);
	 FPT05(startCom:=StepETH=5 ,MODBUS:=MODB06);
	 FPT06(startCom:=StepETH=6 ,MODBUS:=MODB06);
	 FPT07(startCom:=StepETH=7 ,MODBUS:=MODB06);
	 FPT08(startCom:=StepETH=8 ,MODBUS:=MODB06);
	 FPT09(startCom:=StepETH=9 ,MODBUS:=MODB06);
	 FPT10(startCom:=StepETH=10 ,MODBUS:=MODB06); *)

	(*IF StepETH>10 THEN StepETH:=1;END_IF;
	IF NodoDaInterrogareMisuratoreDiPortata_ETH>10 THEN NodoDaInterrogareMisuratoreDiPortata_ETH:=2;END_IF; *)



END_IF


(*==============================*)
(*== System cycle operations ===*)
(*==============================*)
(* Execute TCP processes *)
Logger_Proc();
Remote_Proc();
(*
(* Update user led *)
USRLED_Update();
(* Execute Cron Editor commands *)
*)
END_PROGRAM
ACTION Main_Stm:
CASE Sys.Status OF

	S_STARTUP:
		Sys.Status:=S_INIT_RTC;

	S_INIT_RTC:
		(* Check RTC and update from network *)
		RTC_Update();
		(* Check time *)
		IF Sys.Time_Year>2000 THEN
			Sys.Status:=S_INIT_VAR;
		END_IF








	S_INIT_VAR:
		LogEv(EL_Wrn,EO_SYS,0,1,CONCAT('System_startup_v',WORD_TO_STRING(Plant_SW_VER)));
		Sys.Status:=S_RUNNING;

		OBJ_Definition();


	S_RUNNING:
		Timer1(IN:=NOT Timer1.Q,PT:=T#50ms);
		IF Timer1.Q THEN
			(* Update system checks *)
			SYS_Proc();
		END_IF


		MODB01();

		FOR i:=1 TO Plant_ANZ_INEPRO BY 1 DO
					ANZ_MODBUS_CONNECTOR_INEPRO[i](ModBus:=MODB01);
					ANZ_INEPRO[i](modbusConnector:=ANZ_MODBUS_CONNECTOR_INEPRO[i]);
		END_FOR

		status :=0;
		FOR i:=1 TO Plant_ANZ_INEPRO BY 1 DO IF ANZ_INEPRO[i].Status_Log=1 THEN status :=1;  END_IF	END_FOR

		FOR i:=1 TO Plant_ANZ_INEPRO BY 1 DO IF ANZ_INEPRO[i].Status_Log=2 THEN status :=2;  END_IF	END_FOR






		Timer2(IN:=NOT Timer2.Q,PT:=T#500ms);
		IF Timer2.Q THEN


			(* Read current date/time *)
			RTC_Update();

		(* Letttura ingressi analogici  *)

			PX01	 ( AI_INPUT:=AI_PX01 );
			PX02	 ( AI_INPUT:=AI_PX02 );
			PX03	 ( AI_INPUT:=AI_PX03 );
			PX04	 ( AI_INPUT:=AI_PX04 );





			Lamp( Allarme:=	PX01.Status_Log=2 OR
  						  	PX02.Status_Log=2 OR
  						  	PX03.Status_Log=2 OR
  						  	PX04.Status_Log=2 OR
 						  	COMPRESSORE01.Status_Log=2 OR
						  	COMPRESSORE02.Status_Log=2 OR
						  	COMPRESSORE03.Status_Log=2 OR
						  	COMPRESSORE04.Status_Log=2 OR
							COMPRESSORE05.Status_Log=2 OR
							FPT01.Status_Log=2 OR
							FPT02.Status_Log=2 OR
							FPT03.Status_Log=2 OR
							FPT04.Status_Log=2 OR
							FPT05.Status_Log=2 OR
							FPT06.Status_Log=2 OR
							FPT07.Status_Log=2 OR
							FPT08.Status_Log=2 OR
							FPT09.Status_Log=2 OR
							FPT10.Status_Log=2 OR
							MODB01.Status_Log=2 OR
							MODB02.Status_Log=2 OR
							MODB03.Status_Log=2 OR
							MODB04.Status_Log=2 OR
							MODB05.Status_Log=2
							,
							Warning:=	PX01.Status_Log=1 OR
  						  	PX02.Status_Log=1 OR
  						  	PX03.Status_Log=1 OR
  						  	PX04.Status_Log=1 OR
 						  	COMPRESSORE01.Status_Log=1 OR
						  	COMPRESSORE02.Status_Log=1 OR
						  	COMPRESSORE03.Status_Log=1 OR
						  	COMPRESSORE04.Status_Log=1 OR
							COMPRESSORE05.Status_Log=1 OR
							FPT01.Status_Log=1 OR
							FPT02.Status_Log=1 OR
							FPT03.Status_Log=1 OR
							FPT04.Status_Log=1 OR
							FPT05.Status_Log=1 OR
							FPT06.Status_Log=1 OR
							FPT07.Status_Log=1 OR
							FPT08.Status_Log=1 OR
							FPT09.Status_Log=1 OR
							FPT10.Status_Log=1 OR
							MODB01.Status_Log=1 OR
							MODB02.Status_Log=1 OR
							MODB03.Status_Log=1 OR
							MODB04.Status_Log=1 OR
							MODB05.Status_Log=1
							,
							AllarmeLampada=>LAMP_AL
							);

			(* Test toggle *)
		(*	IF TEST1 THEN TEST1:=FALSE; ELSE TEST1:=TRUE; END_IF*)
		END_IF

		Timer3(IN:=NOT Timer3.Q,PT:=T#5m);
		R_TrigAggiornaLog(clk:=Timer3.Q OR RichiestaDaRemoto OR HMI_AggiornaLog);


		IF R_TrigAggiornaLog.Q THEN
			(* Trig logger *)
		(*	LogTrig(); *)
			EseguiLog:=10;
	     END_IF

	CASE Eseguilog OF

			10 : 	Ton_pausaTrig(IN:=FALSE , PT:=TempoLog , Q=> , ET=> );
					Logger_Head();

					PX01.AddLogData();
					PX02.AddLogData();
					PX03.AddLogData();
					PX04.AddLogData();
					Logger_Send();
					EseguiLog:=20;

			20: Ton_pausaTrig(IN:=TRUE , PT:=TempoLog , Q=> , ET=> );
					IF Ton_pausaTrig.Q THEN
						EseguiLog:=30;
					END_IF

			30 : 	Ton_pausaTrig(IN:=FALSE , PT:=TempoLog , Q=> , ET=> );
					Logger_Head();
					ANZ_INEPRO[1].AddLogData();
					ANZ_INEPRO[2].AddLogData();
					Logger_Send();
					EseguiLog:=40;

			40: Ton_pausaTrig(IN:=TRUE , PT:=TempoLog, Q=> , ET=> );
					IF Ton_pausaTrig.Q THEN
						EseguiLog:=50;
					END_IF

			50 : 	Ton_pausaTrig(IN:=FALSE , PT:=TempoLog , Q=> , ET=> );
					Logger_Head();
					ANZ_INEPRO[3].AddLogData();
					ANZ_INEPRO[4].AddLogData();
					Logger_Send();
					EseguiLog:=60;

			60: Ton_pausaTrig(IN:=TRUE , PT:=TempoLog , Q=> , ET=> );
					IF Ton_pausaTrig.Q THEN
						EseguiLog:=70;
					END_IF
			70 : 	Ton_pausaTrig(IN:=FALSE , PT:=TempoLog , Q=> , ET=> );
					Logger_Head();
					ANZ_INEPRO[5].AddLogData();
					Logger_Send();
					EseguiLog:=80;

			80: Ton_pausaTrig(IN:=TRUE , PT:=TempoLog , Q=> , ET=> );
					IF Ton_pausaTrig.Q THEN
						EseguiLog:=90;
					END_IF
			90 : 	Ton_pausaTrig(IN:=FALSE , PT:=TempoLog , Q=> , ET=> );
					Logger_Head();
					COMPRESSORE01.AddLogData(ModBus:=MODB02);
					COMPRESSORE05.AddLogData(ModBus:=MODB02);
					Logger_Send();
					EseguiLog:=100;

			100: Ton_pausaTrig(IN:=TRUE , PT:=TempoLog , Q=> , ET=> );
					IF Ton_pausaTrig.Q THEN
						EseguiLog:=110;
					END_IF
			110 : 	Ton_pausaTrig(IN:=FALSE , PT:=TempoLog , Q=> , ET=> );
					Logger_Head();
					COMPRESSORE02.AddLogData(ModBus:=MODB03);
					COMPRESSORE03.AddLogData(ModBus:=MODB03);
					COMPRESSORE04.AddLogData(ModBus:=MODB03);
					Logger_Send();
					EseguiLog:=120;

			120: Ton_pausaTrig(IN:=TRUE , PT:=TempoLog , Q=> , ET=> );
					IF Ton_pausaTrig.Q THEN
						EseguiLog:=130;
					END_IF
			130 : 	Ton_pausaTrig(IN:=FALSE , PT:=TempoLog , Q=> , ET=> );
					Logger_Head();
						FPT01.AddLogData(ModBus:=MODB05);
						FPT02.AddLogData();
						FPT03.AddLogData();
						FPT04.AddLogData();
						FPT05.AddLogData();
						FPT06.AddLogData();
						FPT07.AddLogData();
						FPT08.AddLogData();
						FPT09.AddLogData();
						FPT10.AddLogData();

						(*	ESSICATORE01.AddLogData(ModBus:=MODB04); *)
						(*	ESSICATORE02.AddLogData(ModBus:=MODB04); *)
					Logger_Send();
					EseguiLog:=200;



			200: 	RichiestaDaRemoto:=FALSE;


		END_CASE






		Timer4(IN:=NOT Timer4.Q,PT:=T#10s);
		IF Timer4.Q THEN    (* Creo la stringa da salvare  *)
			record:=1;
			IndiceArraRet:=IndiceArraRet+1;

			ArrayDaSalvare[record,IndiceArraRet]:=MID(STR:=sys.Time_LogString, LEN:=8, POS:=3);
			ArrayDaSalvare[record,IndiceArraRet]:=CONCAT(ArrayDaSalvare[record,IndiceArraRet],';');

	(*		ArrayDaSalvare[record,IndiceArraRet]:=WORD_TO_STRING(Sys.Time_Year);
			ArrayDaSalvare[record,IndiceArraRet]:=CONCAT(ArrayDaSalvare[record,IndiceArraRet],BYTE_TO_STRING(Sys.Time_Month));
			ArrayDaSalvare[record,IndiceArraRet]:=CONCAT(ArrayDaSalvare[record,IndiceArraRet],BYTE_TO_STRING(Sys.Time_Day));
		*)	record:=record+1;

			ArrayDaSalvare[record,IndiceArraRet]:=MID(STR:=sys.Time_LogString, LEN:=8, POS:=12);
			ArrayDaSalvare[record,IndiceArraRet]:=CONCAT(ArrayDaSalvare[record,IndiceArraRet],';');

		(*	ArrayDaSalvare[record,IndiceArraRet]:=CONCAT(ArrayDaSalvare[record,IndiceArraRet],'-');
			ArrayDaSalvare[record,IndiceArraRet]:=CONCAT(ArrayDaSalvare[record,IndiceArraRet],MID(STR:=sys.Time_LogString, LEN:=2, POS:=15));
		*)	record:=record+1;

			ArrayDaSalvare[record,IndiceArraRet]:=CONCAT(INT_TO_STRING(PX01.ValoreScalato),';');
			record:=record+1;
			ArrayDaSalvare[record,IndiceArraRet]:=CONCAT(INT_TO_STRING(PX02.ValoreScalato),';');
			record:=record+1;
			ArrayDaSalvare[record,IndiceArraRet]:=CONCAT(INT_TO_STRING(PX03.ValoreScalato),';');
			record:=record+1;
			ArrayDaSalvare[record,IndiceArraRet]:=CONCAT(INT_TO_STRING(PX04.ValoreScalato),';');
			record:=record+1;

			ArrayDaSalvare[record,IndiceArraRet]:=CONCAT(REAL_TO_STRING(DWORD_TO_REAL(FPT01.Parametro18)/10),';');
			record:=record+1;
			ArrayDaSalvare[record,IndiceArraRet]:=CONCAT(REAL_TO_STRING(INT_TO_REAL(FPT01.IntPressioneCalcolata)/10),';');
			record:=record+1;
			ArrayDaSalvare[record,IndiceArraRet]:=CONCAT(REAL_TO_STRING(DWORD_TO_REAL(FPT01.Parametro128)/10),';');
			record:=record+1;

			ArrayDaSalvare[record,IndiceArraRet]:=CONCAT(REAL_TO_STRING(DWORD_TO_REAL(FPT02.Parametro18)/10),';');
			record:=record+1;
			ArrayDaSalvare[record,IndiceArraRet]:=CONCAT(REAL_TO_STRING(DWORD_TO_REAL(FPT02.IntPressioneCalcolata)/10),';');
			record:=record+1;
			ArrayDaSalvare[record,IndiceArraRet]:=CONCAT(REAL_TO_STRING(DWORD_TO_REAL(FPT02.Parametro128)/10),';');
			record:=record+1;

			ArrayDaSalvare[record,IndiceArraRet]:=CONCAT(REAL_TO_STRING(DWORD_TO_REAL(FPT03.Parametro18)/10),';');
			record:=record+1;
			ArrayDaSalvare[record,IndiceArraRet]:=CONCAT(REAL_TO_STRING(DWORD_TO_REAL(FPT03.IntPressioneCalcolata)/10),';');
			record:=record+1;
			ArrayDaSalvare[record,IndiceArraRet]:=CONCAT(REAL_TO_STRING(DWORD_TO_REAL(FPT03.Parametro128)/10),';');
			record:=record+1;

			ArrayDaSalvare[record,IndiceArraRet]:=CONCAT(REAL_TO_STRING(DWORD_TO_REAL(FPT04.Parametro18)/10),';');
			record:=record+1;
			ArrayDaSalvare[record,IndiceArraRet]:=CONCAT(REAL_TO_STRING(DWORD_TO_REAL(FPT04.IntPressioneCalcolata)/10),';');
			record:=record+1;
			ArrayDaSalvare[record,IndiceArraRet]:=CONCAT(REAL_TO_STRING(DWORD_TO_REAL(FPT04.Parametro128)/10),';');
			record:=record+1;

			ArrayDaSalvare[record,IndiceArraRet]:=CONCAT(REAL_TO_STRING(DWORD_TO_REAL(FPT05.Parametro18)/10),';');
			record:=record+1;
			ArrayDaSalvare[record,IndiceArraRet]:=CONCAT(REAL_TO_STRING(DWORD_TO_REAL(FPT05.IntPressioneCalcolata)/10),';');
			record:=record+1;
			ArrayDaSalvare[record,IndiceArraRet]:=CONCAT(REAL_TO_STRING(DWORD_TO_REAL(FPT05.Parametro128)/10),';');
			record:=record+1;

			ArrayDaSalvare[record,IndiceArraRet]:=CONCAT(REAL_TO_STRING(DWORD_TO_REAL(FPT06.Parametro18)/10),';');
			record:=record+1;
			ArrayDaSalvare[record,IndiceArraRet]:=CONCAT(REAL_TO_STRING(DWORD_TO_REAL(FPT06.IntPressioneCalcolata)/10),';');
			record:=record+1;
			ArrayDaSalvare[record,IndiceArraRet]:=CONCAT(REAL_TO_STRING(DWORD_TO_REAL(FPT06.Parametro128)/10),';');
			record:=record+1;

			ArrayDaSalvare[record,IndiceArraRet]:=CONCAT(REAL_TO_STRING(DWORD_TO_REAL(FPT07.Parametro18)/10),';');
			record:=record+1;
			ArrayDaSalvare[record,IndiceArraRet]:=CONCAT(REAL_TO_STRING(DWORD_TO_REAL(FPT07.IntPressioneCalcolata)/10),';');
			record:=record+1;
			ArrayDaSalvare[record,IndiceArraRet]:=CONCAT(REAL_TO_STRING(DWORD_TO_REAL(FPT07.Parametro128)/10),';');
			record:=record+1;

			ArrayDaSalvare[record,IndiceArraRet]:=CONCAT(REAL_TO_STRING(DWORD_TO_REAL(FPT08.Parametro18)/10),';');
			record:=record+1;
			ArrayDaSalvare[record,IndiceArraRet]:=CONCAT(REAL_TO_STRING(DWORD_TO_REAL(FPT08.IntPressioneCalcolata)/10),';');
			record:=record+1;
			ArrayDaSalvare[record,IndiceArraRet]:=CONCAT(REAL_TO_STRING(DWORD_TO_REAL(FPT08.Parametro128)/10),';');
			record:=record+1;

			ArrayDaSalvare[record,IndiceArraRet]:=CONCAT(REAL_TO_STRING(DWORD_TO_REAL(FPT09.Parametro18)/10),';');
			record:=record+1;
			ArrayDaSalvare[record,IndiceArraRet]:=CONCAT(REAL_TO_STRING(DWORD_TO_REAL(FPT09.IntPressioneCalcolata)/10),';');
			record:=record+1;
			ArrayDaSalvare[record,IndiceArraRet]:=CONCAT(REAL_TO_STRING(DWORD_TO_REAL(FPT09.Parametro128)/10),';');
			record:=record+1;

			ArrayDaSalvare[record,IndiceArraRet]:=CONCAT(REAL_TO_STRING(DWORD_TO_REAL(FPT10.Parametro18)/10),';');
			record:=record+1;
			ArrayDaSalvare[record,IndiceArraRet]:=CONCAT(REAL_TO_STRING(DWORD_TO_REAL(FPT10.IntPressioneCalcolata)/10),';');
			record:=record+1;
			ArrayDaSalvare[record,IndiceArraRet]:=CONCAT(REAL_TO_STRING(DWORD_TO_REAL(FPT10.Parametro128)/10),';');
			record:=record+1;

			ArrayDaSalvare[record,IndiceArraRet]:=CONCAT(REAL_TO_STRING(INT_TO_REAL(ESSICATORE02.Probe1)/10),';');
			record:=record+1;
			ArrayDaSalvare[record,IndiceArraRet]:=CONCAT('---',';');
			record:=record+1;


			ArrayDaSalvare[record,IndiceArraRet]:=CONCAT((SEL(COMPRESSORE01.StatusControl[2],'LOAD','UNLOAD')),';');
			record:=record+1;
			ArrayDaSalvare[record,IndiceArraRet]:=CONCAT(REAL_TO_STRING(INT_TO_REAL(COMPRESSORE01.MB_RegistriHoldingLetti[3])/10),';');
			record:=record+1;
			ArrayDaSalvare[record,IndiceArraRet]:=CONCAT(REAL_TO_STRING(INT_TO_REAL(COMPRESSORE01.MB_RegistriHoldingLetti[20])/1),';');
			record:=record+1;
			ArrayDaSalvare[record,IndiceArraRet]:=CONCAT(REAL_TO_STRING(INT_TO_REAL(COMPRESSORE01.MB_RegistriHoldingLetti[112])/10),';');
			record:=record+1;
			ArrayDaSalvare[record,IndiceArraRet]:=CONCAT(REAL_TO_STRING(INT_TO_REAL(COMPRESSORE01.MB_RegistriHoldingLetti[113])/10),';');
			record:=record+1;
			ArrayDaSalvare[record,IndiceArraRet]:=CONCAT(REAL_TO_STRING(INT_TO_REAL(COMPRESSORE01.MB_RegistriHoldingLetti[114])/10),';');
			record:=record+1;

			ArrayDaSalvare[record,IndiceArraRet]:=CONCAT(SEL(COMPRESSORE02.StatusControl[2],'LOAD','UNLOAD'),';');
			record:=record+1;
			ArrayDaSalvare[record,IndiceArraRet]:=CONCAT(REAL_TO_STRING(INT_TO_REAL(COMPRESSORE02.MB_RegistriHoldingLetti[3])/10),';');
			record:=record+1;
			ArrayDaSalvare[record,IndiceArraRet]:=CONCAT(REAL_TO_STRING(INT_TO_REAL(COMPRESSORE02.MB_RegistriHoldingLetti[20])/1),';');
			record:=record+1;
			ArrayDaSalvare[record,IndiceArraRet]:=CONCAT(REAL_TO_STRING(INT_TO_REAL(COMPRESSORE02.MB_RegistriHoldingLetti[112])/10),';');
			record:=record+1;
			ArrayDaSalvare[record,IndiceArraRet]:=CONCAT(REAL_TO_STRING(INT_TO_REAL(COMPRESSORE02.MB_RegistriHoldingLetti[113])/10),';');
			record:=record+1;
			ArrayDaSalvare[record,IndiceArraRet]:=CONCAT(REAL_TO_STRING(INT_TO_REAL(COMPRESSORE02.MB_RegistriHoldingLetti[130])/10),';');
			record:=record+1;

			ArrayDaSalvare[record,IndiceArraRet]:=CONCAT(SEL(COMPRESSORE03.StatusControl[2],'LOAD','UNLOAD'),';');
			record:=record+1;
			ArrayDaSalvare[record,IndiceArraRet]:=CONCAT(REAL_TO_STRING(INT_TO_REAL(COMPRESSORE03.MB_RegistriHoldingLetti[3])/10),';');
			record:=record+1;
			ArrayDaSalvare[record,IndiceArraRet]:=CONCAT(REAL_TO_STRING(INT_TO_REAL(COMPRESSORE03.MB_RegistriHoldingLetti[20])/1),';');
			record:=record+1;
			ArrayDaSalvare[record,IndiceArraRet]:=CONCAT(REAL_TO_STRING(INT_TO_REAL(COMPRESSORE03.MB_RegistriHoldingLetti[112])/10),';');
			record:=record+1;
			ArrayDaSalvare[record,IndiceArraRet]:=CONCAT(REAL_TO_STRING(INT_TO_REAL(COMPRESSORE03.MB_RegistriHoldingLetti[113])/10),';');
			record:=record+1;
			ArrayDaSalvare[record,IndiceArraRet]:=CONCAT(REAL_TO_STRING(INT_TO_REAL(COMPRESSORE03.MB_RegistriHoldingLetti[130])/10),';');
			record:=record+1;

			ArrayDaSalvare[record,IndiceArraRet]:=CONCAT(SEL(COMPRESSORE04.StatusControl[2],'LOAD','UNLOAD'),';');
			record:=record+1;
			ArrayDaSalvare[record,IndiceArraRet]:=CONCAT(REAL_TO_STRING(INT_TO_REAL(COMPRESSORE04.MB_RegistriHoldingLetti[3])/10),';');
			record:=record+1;
			ArrayDaSalvare[record,IndiceArraRet]:=CONCAT(REAL_TO_STRING(INT_TO_REAL(COMPRESSORE04.MB_RegistriHoldingLetti[20])/1),';');
			record:=record+1;
			ArrayDaSalvare[record,IndiceArraRet]:=CONCAT(REAL_TO_STRING(INT_TO_REAL(COMPRESSORE04.MB_RegistriHoldingLetti[112])/10),';');
			record:=record+1;
			ArrayDaSalvare[record,IndiceArraRet]:=CONCAT(REAL_TO_STRING(INT_TO_REAL(COMPRESSORE04.MB_RegistriHoldingLetti[113])/10),';');
			record:=record+1;
			ArrayDaSalvare[record,IndiceArraRet]:=CONCAT(REAL_TO_STRING(INT_TO_REAL(COMPRESSORE04.MB_RegistriHoldingLetti[130])/10),';');
			record:=record+1;

			ArrayDaSalvare[record,IndiceArraRet]:=CONCAT(SEL(COMPRESSORE05.StatusControl[2],'LOAD','UNLOAD'),';');
			record:=record+1;
			ArrayDaSalvare[record,IndiceArraRet]:=CONCAT(REAL_TO_STRING(INT_TO_REAL(COMPRESSORE05.MB_RegistriHoldingLetti[3])/10),';');
			record:=record+1;
			ArrayDaSalvare[record,IndiceArraRet]:=CONCAT(REAL_TO_STRING(INT_TO_REAL(COMPRESSORE05.MB_RegistriHoldingLetti[20])/1),';');
			record:=record+1;
			ArrayDaSalvare[record,IndiceArraRet]:=CONCAT(REAL_TO_STRING(INT_TO_REAL(COMPRESSORE05.MB_RegistriHoldingLetti[112])/10),';');
			record:=record+1;
			ArrayDaSalvare[record,IndiceArraRet]:=CONCAT(REAL_TO_STRING(INT_TO_REAL(COMPRESSORE05.MB_RegistriHoldingLetti[113])/10),';');
			record:=record+1;
			ArrayDaSalvare[record,IndiceArraRet]:=CONCAT(REAL_TO_STRING(INT_TO_REAL(COMPRESSORE05.MB_RegistriHoldingLetti[130])/10),';');

			IF IndiceArraRet>=60 THEN

				CreaFile(IndiceArray:= IndiceArraRet,NumRecord:=record);

				FOR k:=0 TO IndiceArraRet DO
					FOR x:=0 TO record DO
					ArrayDaSalvare[k,x]:='';
					END_FOR
				END_FOR

				IndiceArraRet:=0;
			END_IF

	END_IF




	S_SHUTDOWN:
		(* Stop caldaia *)
		(* Stop deviatori *)
		(* Aspetta 5 min prima di spegnere eventuali circolatori *)
		Sys.Status:=S_STARTUP;

	S_HALT:
		(* Aspetta uscita manuale *)
		Sys.Status:=S_STARTUP;


ELSE
	Sys.Status:=S_STARTUP;
END_CASE;
END_ACTION
ACTION OBJ_Definition:
(**** Define Plant Objects ****)

ANZ_INEPRO_DefineRegisters();

FOR I:=1 TO Plant_ANZ_INEPRO DO
	ANZ_INEPRO[i].ID := i;
	ANZ_INEPRO[i].TIMING_AGGREGATED_MEASURE:=ANZ_INEPRO_POLLING_TIME;
	ANZ_INEPRO[i].TIMING_RESET_AGGREGATED_MEASURE:=t#15m;
	ANZ_MODBUS_CONNECTOR_INEPRO [i].PARENT_EO_TYPE := EO_ANZ;
	ANZ_MODBUS_CONNECTOR_INEPRO [i].PARENT_EO_ID := i;
	ANZ_MODBUS_CONNECTOR_INEPRO [i].Address := i;
	ANZ_MODBUS_CONNECTOR_INEPRO [i].TIMING:=ANZ_INEPRO_POLLING_TIME+WORD_TO_TIME(ANZ_INEPRO[i].ID*1000);
	ANZ_MODBUS_CONNECTOR_INEPRO [i].retryErrMax:=10;

END_FOR
END_ACTION

(* POU Plant_Objects/obj_CreaFile, ST *)
FUNCTION_BLOCK obj_CreaFile
VAR_INPUT
	(*StringaDaScrivere:STRING(180); *)
	IndiceArray:INT;
	NumRecord:INT;

END_VAR

VAR

	hFile: 	DWORD;
	nFile: 	DWORD;
	IntestazioneArray: ARRAY [0..80] OF STRING(20) :='Data;','ORA;',
													'PT401.bar;' , 'PT301.bar;','PT104.bar;','PT101.bar;',
													'FT102.m3 n/hr;','FT102.barg;','FT102.m3 n/hr;',
													'FT103.n/hr;','FT103.barg;','FT103.m3 n/hr;',
													'FT201.m3n/hr;','FT201.barg;','FT201.m3 n/hr;',
													'FT302.m3n/hr;','FT302.barg;','FT302.m3 n/hr;',
													'FT402.m3n/hr;','FT402.barg;','FT402.m3 n/hr;',
													'FT203.m3n/hr;','FT203.barg;','FT203.m3 n/hr;',
													'FT303.m3n/hr;','FT303.barg;','FT303.m3 n/hr;',
													'FT304.m3n/hr;','FT304.barg;','FT304.m3 n/hr;',
													'FT305.m3n/hr;','FT305.barg;','FT305.m3 n/hr;',
													'FT403.m3n/hr;','FT403.barg;','FT403.m3 n/hr;',
													'E102.°C;','E102.°C;',
													'C101.Load/Unload;','C101.DP_barg;','C101.%;','C101.TP_barg;','C101.ASP_barg;','C101.ISP_barg;',
													'C102.Load/Unload;','C102.DP_barg;','C102.%;','C102.TP_barg;','C102.ASP_barg;','C102.ISP_barg;',
													'C103.Load/Unload;','C103.DP_barg;','C103.%;','C103.TP_barg;','C103.ASP_barg;','C103.ISP_barg;',
													'C104.Load/Unload;','C104.DP_barg;','C104.%;','C104.TP_barg;','C104.ASP_barg;','C104.ISP_barg;',
													'C105.Load/Unload;','C105.DP_barg;','C105.%;','C105.TP_barg;','C105.ASP_barg;','C105.ISP_barg;'
													;

(*	Intestazione:STRING(500);
	StringaDaScrivere:STRING(500); *)
	x: INT;
(*	Minute: STRING;
	Hour: STRING; *)

	FineLinea: STRING:='$R$N';

	k: INT;
	CheckSpazio: GET_STATUS_VOLUME;
	SpazioLibero: UDINT;
	SpazioSD: UDINT;
	ErroreSpazio: BOOL;
	fALARM_ErroreSpazio		:FLT_TAP;


END_VAR

VAR RETAIN
	GiornoSalvato: BYTE;
	LogFileName:STRING;
END_VAR
(* Check spazio Micor SD *)

CheckSpazio(VOLUME:='S:\' , ERRCODE=> , FREE=>SpazioLibero , TOTAL=>SpazioSD );

IF SpazioLibero<10000 THEN

	ErroreSpazio:=TRUE;

ELSE

	ErroreSpazio:=FALSE;


	IF (Sys.Time_Day) <> GiornoSalvato THEN
		GiornoSalvato:=(Sys.Time_Day);

		LogFileName:='S:\';
		LogFileName:=CONCAT(LogFileName,MID(STR:=sys.Time_LogString, LEN:=10, POS:=1));


	(*	LogFileName:=CONCAT(LogFileName,BYTE_TO_STRING(Sys.Time_Month));
		LogFileName:=CONCAT(LogFileName,BYTE_TO_STRING(Sys.Time_Day));*)

	(*	Hour:=MID(STR:=sys.Time_LogString, LEN:=2, POS:=12);
		Minute:=MID(STR:=sys.Time_LogString, LEN:=2, POS:=15);

		LogFileName:=CONCAT(LogFileName,Hour);
		LogFileName:=CONCAT(LogFileName,Minute);  *)
		LogFileName:=CONCAT(LogFileName,'.csv');

		hFile:=SysFileOpen(LogFileName,'r');

		IF hFile=0 THEN
			(*** Creo il fiel se non esiste *)
			hFile:=SysFileOpen(LogFileName,'w');
			IF hFile<>0 THEN
				FOR x:=0 TO NumRecord DO
					SysFileWrite(hFile,ADR( IntestazioneArray[x]),LEN(IntestazioneArray[x]));
				END_FOR
			      		SysFileWrite(hFile, ADR(FineLinea), LEN(FineLinea));

				FOR x:=1 TO IndiceArray   DO
					FOR k:=0 TO NumRecord  DO
						SysFileWrite(hFile,ADR( (PLC_PRG.ArrayDaSalvare[k,x])),LEN((PLC_PRG.ArrayDaSalvare[k,x])));
					END_FOR
					SysFileWrite(nFile, ADR(FineLinea), LEN(FineLinea));
				END_FOR
			END_IF
			SysFileClose(hFile);
		ELSE
			SysFileClose(hFile);
		END_IF

	ELSE


		nFile:=SysFileOpen(LogFileName,'a');
		IF nFile<>0 THEN
			FOR x:=1 TO IndiceArray DO
				FOR k:=0 TO NumRecord  DO
					SysFileWrite(hFile,ADR( (PLC_PRG.ArrayDaSalvare[k,x])),LEN((PLC_PRG.ArrayDaSalvare[k,x])));
				END_FOR
				SysFileWrite(nFile, ADR(FineLinea), LEN(FineLinea));
			END_FOR
			SysFileClose(nFile);
		END_IF
	END_IF


END_IF


fALARM_ErroreSpazio(IN:=Errorespazio OR (CheckSpazio.ERRCODE<>0));
IF fALARM_ErroreSpazio.EVH THEN
	LogEv(EL_Wrn,EO_SYS,0,1,'Memoria_SD_Piena');
END_IF
IF fALARM_ErroreSpazio.EVL THEN
	LogEv(EL_Log,EO_SYS,0,1,'Memoria_SD_Libera');
END_IF
END_FUNCTION_BLOCK

(* POU Utils Functions/FLT_TAP, ST *)
FUNCTION_BLOCK FLT_TAP
VAR_INPUT
	IN		: BOOL;
	TAP		: BYTE:=4;
	INITEV	: BOOL:=TRUE;
END_VAR
VAR_OUTPUT
	OUT		: BOOL;
	EVH		: BOOL;
	EVL		: BOOL;
END_VAR
VAR
	init	: BOOL:=FALSE;
	cnt		: BYTE;
END_VAR
EVH:=FALSE;
EVL:=FALSE;

IF NOT init THEN
	init := TRUE;
	IF INITEV THEN
		OUT  := NOT IN;
		cnt  := TAP;
	ELSE
		OUT  := IN;
	END_IF
END_IF

IF OUT<>IN THEN
	cnt:=cnt+1;
	IF cnt>TAP THEN
		OUT:=IN;
		cnt:=0;
		IF OUT THEN EVH:=TRUE; ELSE EVL:=TRUE; END_IF
	END_IF
ELSE
	cnt:=0;
END_IF
END_FUNCTION_BLOCK

(* POU TCP_Logger/LogEv, ST *)
FUNCTION LogEv : BOOL
VAR_INPUT
	Level	: en_Logger_ErrLev;
	Object  : en_SYS_Objects;
	Index	: WORD;
	Error	: WORD;
	Message : STRING;
END_VAR
VAR
	s1 : STRING(160);
	i  : INT;
END_VAR
(* Execute error level operations *)

Sys.Alarm:=Lamp.SistemaInAllarme;
Sys.Warning:=Lamp.SistemaWarning;


(* Fill lastlog list *)
s1:=CONCAT(Sys.Time_LogString,';Lev=');
s1:=CONCAT(s1,INT_TO_STRING(Level));
s1:=CONCAT(s1,';Obj=');
s1:=CONCAT(s1,INT_TO_STRING(Object));
s1:=CONCAT(s1,';Idx=');
s1:=CONCAT(s1,WORD_TO_STRING(Index));
s1:=CONCAT(s1,';Err=');
s1:=CONCAT(s1,WORD_TO_STRING(Error));
Sys.LastLogs_Dat[Sys.LastLogs_Idx]:=s1;
Sys.LastLogs_Msg[Sys.LastLogs_Idx]:=Message;
Sys.LastLogs_Idx:=Sys.LastLogs_Idx+1;
IF Sys.LastLogs_Idx>5 THEN Sys.LastLogs_Idx:=0; END_IF

(*---------------------------------------------------------------*)
	Logger_Head();
(*---------------------------------------------------------------*)

(* Insert ERR *)
s1:=CONCAT('&ERR=',INT_TO_STRING(Level));
s1:=CONCAT(s1,';');
s1:=CONCAT(s1,INT_TO_STRING(Object));
s1:=CONCAT(s1,';');
s1:=CONCAT(s1,WORD_TO_STRING(Index));
s1:=CONCAT(s1,';');
s1:=CONCAT(s1,WORD_TO_STRING(Error));
s1:=CONCAT(s1,';');
ADDSTRING(ADR(Logger.TData), ADR(s1), Logger.TLen);
s1:=Message;
STR_NOSPACES(ADR(s1));
ADDSTRING(ADR(Logger.TData), ADR(s1), Logger.TLen);

(*---------------------------------------------------------------*)
	Logger_Send();
(*---------------------------------------------------------------*)
END_FUNCTION

(* POU TCP_Logger/Logger_Head, ST *)
FUNCTION Logger_Head : BOOL
VAR
	s1 : STRING(160);
	i  : BYTE;
END_VAR
Logger.TLen:=0;
(* Set GET header *)
ADDSTRING(ADR(Logger.TData), ADR(Logger_GETSTART), Logger.TLen);

(* Insert Header *)
s1:=INSERT('ID=&V=1&D=',DWORD_TO_STRING(Plant_SN),3);
s1:=CONCAT(s1,REPLACE(Sys.Time_LogString,'T',1,11));
(*s1:=CONCAT(s1,Sys.Time_LogString) *)
s1:=CONCAT(s1,'&S=');
IF Sys.Alarm THEN i:=2; ELSIF Sys.Warning THEN i:=1; ELSE i:=0; END_IF
s1:=CONCAT(s1,BYTE_TO_STRING(i));
ADDSTRING(ADR(Logger.TData), ADR(s1), Logger.TLen);
END_FUNCTION

(* POU Utils Functions/ADDSTRING, ST *)
FUNCTION ADDSTRING : BOOL
VAR_INPUT
	pTxData: POINTER TO BYTE;
	pString: POINTER TO BYTE;
END_VAR
VAR_IN_OUT
	TxLen: DINT;
END_VAR
VAR
END_VAR
pTxData:=pTxData+TxLen;
WHILE pString^<>0 DO
	pTxData^:=pString^;
	pString:=pString+1;
	pTxData:=pTxData+1;
	TxLen:=TxLen+1;
END_WHILE
END_FUNCTION

(* POU Utils Functions/STR_NOSPACES, ST *)
FUNCTION STR_NOSPACES : BOOL (* Replace spaces and bad chars with allowed ones, used as HTTP-GET validator *)
VAR_INPUT
	pString: POINTER TO BYTE;
END_VAR
VAR
END_VAR
WHILE pString^<>0 DO
	IF pString^=16#20 (* space *) THEN pString^:=16#5F; (*'_'*) END_IF
	pString:=pString+1;
END_WHILE
END_FUNCTION

(* POU TCP_Logger/Logger_Send, ST *)
FUNCTION Logger_Send : BOOL
VAR
	hFile: 	DWORD;
	pos:	DWORD;
END_VAR
(* Finalize string *)
ADDSTRING(ADR(Logger.TData), ADR(Logger_GETEND), Logger.TLen);

(* Read log position *)
pos:=SysFileGetSize(Logger_DataFile);
(* Check log size, bckup and erase if no pending messages *)
IF pos>5000000(*5M*) THEN
	hFile:=SysFileOpen(Logger_IndexFile,'r');
	IF hFile=0 THEN
		SysFileDelete(Logger_DataFileOld);
		SysFileRename(Logger_DataFile,Logger_DataFileOld);
		pos:=0;
	ELSE
		SysFileClose(hFile);
	END_IF
END_IF
(* Write message on log file *)
hFile:=SysFileOpen(Logger_DataFile,'a');
IF hFile<>0 THEN
	SysFileWrite(hFile, ADR(Logger.TData), Logger.TLen);
	SysFileClose(hFile);
ELSE
	Sys.Warning:=TRUE;
END_IF


(* Check logger status *)
IF Logger.SendReq=FALSE THEN
	(* Set log position for recovery *)
	Logger.SendIdx:=pos;
	(* Copy message data *)
	MEMCPY(ADR(Logger.TData),ADR(Logger.SendData),DINT_TO_WORD(Logger.TLen));
	Logger.SendLen:=Logger.TLen;
	(* Trigger request *)
	Logger.SendReq:=TRUE;
ELSE
	(* Add message position+size in recovery indexes *)
	hFile:=SysFileOpen(Logger_IndexFile,'a');
	SysFileWrite(hFile, ADR(pos), SIZEOF(pos));
	SysFileWrite(hFile, ADR(Logger.TLen), SIZEOF(Logger.TLen));
	SysFileClose(hFile);
END_IF
END_FUNCTION

(* POU Utils Functions/MEMCPY, ST *)
FUNCTION MEMCPY:BOOL
VAR_INPUT
	pSourceAddress:POINTER TO ARRAY[1..2] OF BYTE;
	pDestinationAddress:POINTER TO ARRAY[1..2] OF BYTE;
	BytesToCopy:WORD;
END_VAR
VAR
END_VAR
WHILE (BytesToCopy > 0) DO
	pDestinationAddress^[1]:=pSourceAddress^[1]; (* copy bytes from source to destination *)
	pDestinationAddress:=ADR(pDestinationAddress^[2]); (* increment destination *)
	pSourceAddress:=ADR(pSourceAddress^[2]);(* increment source *)
	BytesToCopy:=BytesToCopy -1; (* decrement number of bytes to copy *)
END_WHILE
END_FUNCTION

(* POU TCP_Logger/Logger_Proc, ST *)
PROGRAM Logger_Proc
VAR
	c1:         	TCPCLIENT;

	Open:	    	BOOL;
	IpAddr:			DWORD;
	InetAddr:		DWORD;
	Connected:  	BOOL;
	Error:      	DINT;
	TxTrig:     	BOOL;
	RxData:			ARRAY [0..MAX_RECEIVE_TCP_CLIENT] OF BYTE;
	RxLen:			DINT;

	Retry:			BYTE;	(* Counter for connection retries *)
	Recovered:		BYTE;	(* Counter for recovered unsent messages *)

	i:				DINT;
	pos:			DWORD;
	hFile:			DWORD;

END_VAR
(*=== State machine ===*)
CASE Logger.Status OF

	S_Logger_UNKNOWN:
		(* Startup *)
		Logger.SendReq:=FALSE;
		Open:=FALSE;
		Logger.Status:=S_Logger_IDLE;

	S_Logger_IDLE:
		(* Wait request *)
		IF Logger.SendReq THEN
			(* Resolve server name or use static IP *)
			IF LEN(Logger_SERVER)=0 THEN
				InetAddr:=SysSockInetAddr(Logger_IP);
			ELSE
				IpAddr:=SysSockGetHostByName(ADR(Logger_SERVER));
				DWORDSWAP(pIn:=ADR(IpAddr), pOut:=ADR(InetAddr));
			END_IF
			TxTrig:=FALSE;
			RxLen:=0;
			(* Open connection *)
			Open:=TRUE;
			Logger.Status:=S_Logger_WAITCONN;
		END_IF

	S_Logger_WAITCONN:
		(* Wait connection *)
		IF Connected THEN
			(* Send data *)
			TxTrig:=TRUE;
			Logger.Status:=S_Logger_WAITTX;
		END_IF
		IF Error>0 THEN
			Open:=FALSE;
			Logger.Status:=S_Logger_ERROR;
		END_IF

	S_Logger_WAITTX:
		(* Wait transmission *)
		IF NOT TxTrig THEN
			Logger.Status:=S_Logger_WAITRESP;
		END_IF
		IF Error>0 THEN
			Open:=FALSE;
			Logger.Status:=S_Logger_ERROR;
		END_IF

	S_Logger_WAITRESP:
		(* Wait response *)
		IF Connected=FALSE (* OR TIMEOUT!! *) THEN
			Open:=FALSE;
			(* Check response *)
			IF RxLen>=4 AND CHKSTRING(pString:=ADR(RxData), pPattern:=ADR(Logger_CHECK)) THEN
				Logger.SendReq:=FALSE;
				Retry:=0;
				(* Check unsent messages to flush *)
				IF Recovered<Logger_RecoverMsgs THEN
					MsgChk();
					IF Logger.SendReq=TRUE THEN
						Recovered:=Recovered+1;
					ELSE
						Recovered:=0;
					END_IF
				ELSE
					Recovered:=0;
				END_IF
				Logger.Status:=S_Logger_IDLE;
			ELSE
				Logger.Status:=S_Logger_ERROR;
			END_IF
		END_IF

	S_Logger_ERROR:
		(* Connection error or send failure *)
		Retry:=Retry+1;
		IF Retry>Logger_ConnRetries THEN
			(* Save message as unsent *)
			MsgSave();
			Logger.SendReq:=FALSE;
			Retry:=0;
		END_IF
		Logger.Status:=S_Logger_IDLE;

ELSE
	Logger.Status:=S_Logger_UNKNOWN;
END_CASE


(*=== Execute client lib ===*)
c1(
	xOpenConnection			:= Open,
	dwInetAddr 				:= InetAddr,
	wPortNumber				:= Logger_PORT,
	ptSendData				:= ADR(Logger.SendData),
	diSendCount				:= Logger.SendLen,
	tConnectWatchdogTime	:= t#10s,
	xStartSend				:= TxTrig,
	aReceiveBuffer			:= RxData,
	diReceiveCount			:= RxLen,
	xConnected				=> Connected,
	diError					=> Error
);

(*=== Process Rx data ===*)
(*IF RxLen>0 THEN
	RxLen:=0;
END_IF*)
END_PROGRAM
ACTION MsgChk:
(* Open index file *)
hFile:=SysFileOpen(Logger_IndexFile,'r');
IF hFile=0 THEN
	RETURN;
END_IF
(* Search oldest message to recover *)
SysFileSetPos(hFile,Logger.LastIdxPos);
Logger.SendLen:=0;
REPEAT
	SysFileRead(hFile, ADR(Logger.SendIdx), SIZEOF(Logger.SendIdx));
	pos:=SysFileGetPos(hFile);
	SysFileRead(hFile, ADR(Logger.SendLen), SIZEOF(Logger.SendLen));
UNTIL
	SysFileEOF(hFile) OR Logger.SendLen<>0
END_REPEAT
SysFileClose(hFile);
(* Delete index file when all messages are recovered *)
IF Logger.SendLen=0 THEN
	Logger.LastIdxPos:=0;
	SysFileDelete(Logger_IndexFile);
	RETURN;
END_IF
(* Recover message data *)
hFile:=SysFileOpen(Logger_DataFile,'r');
IF hFile<>0 THEN
	SysFileSetPos(hFile,Logger.SendIdx);
	SysFileRead(hFile,ADR(Logger.SendData),Logger.SendLen);
	Logger.SendReq:=TRUE;
	SysFileClose(hFile);
END_IF
(* Clear index entry *)
hFile:=SysFileOpen(Logger_IndexFile,'a');
IF hFile<>0 THEN
	SysFileSetPos(hFile,pos);
	i:=0;
	SysFileWrite(hFile, ADR(i), 4);
	Logger.LastIdxPos:=SysFileGetPos(hFile);
	SysFileClose(hFile);
END_IF
END_ACTION
ACTION MsgSave:
(* Add log position in recovery indexes *)
hFile:=SysFileOpen(Logger_IndexFile,'a');
SysFileWrite(hFile, ADR(Logger.SendIdx), SIZEOF(Logger.SendIdx));
SysFileWrite(hFile, ADR(Logger.SendLen), SIZEOF(Logger.SendLen));
SysFileClose(hFile);
END_ACTION

(* POU Utils Functions/TCPCLIENT, ST *)
FUNCTION_BLOCK TCPCLIENT
(***********************************************************************************************************	*)
(* Version: 1.3b                        			          													*)
(* Date: 28.10.2014                   				          							            			*)
(***********************************************************************************************************	*)
(* WAGO Kontakttechnik GmbH Hansastr. 27 32423 Minden(Westf.)													*)
(* Tel. +0049 571/887-0 Fax. +0049 571/887-0																	*)
(* Author: VB																									*)
(***********************************************************************************************************	*)
(*Description:	A TCP client to read and write data with additional connection watchdog							*)
(*History:																										*)
(*Version 1.3b: 28.10.2014: Use DWORD address for IP (Andrea Ravasio)											*)
(*Version 1.3: 11.02.2011: Changes according to 750-880/881											 			*)
(*Version 1.2: 29.08.2007 Bugfix TCP Client																		*)
(*Version 1.1: 15.01.2007 Changes according to FW11																*)
(*Version 1.0: 09.03.2006 Release																				*)
(***********************************************************************************************************	*)
VAR CONSTANT
	STATE_CREATE     				 : BYTE:= 0;
	STATE_OPEN     					 : BYTE:= 1;
	STATE_IOCTL    					 : BYTE:= 2;
	STATE_CONNECT     				 : BYTE:= 10;
	STATE_TX       					 : BYTE:= 20;
	STATE_RX       					 : BYTE:= 30;
	STATE_CLOSE    					 : BYTE:= 40;
	STATE_ERROR_TRAP			     : BYTE:= 200;
END_VAR

VAR_INPUT
	xOpenConnection					: BOOL;
	dwInetAddr						: DWORD; (* <== Use SysSockInetAddr() value or
													swapped bytes order of SysSockGetHostByName() value *)
	wPortNumber						: WORD;
	ptSendData						: POINTER TO ARRAY[0..MAX_SEND_TCP_CLIENT] OF BYTE;
	diSendCount						: DINT;
	tConnectWatchdogTime		    : TIME := t#10s;
END_VAR
VAR_OUTPUT
	xConnected						: BOOL;
	diError 						: DINT := 0;
END_VAR
(* ErrorCodes -----------------------------------------
	16#8001 => No socket descriptor available 
	16#8002 => SysSockSend returns -1 
	16#8003 => Socket was "gracefully closed" 
	16#8004 => switching to none blocking mode fails
	16#8005 => SysSockClose() returns FALSE 
    16#8006 => SysSockConnect() fails
    16#8007 => SysSockSend() fails
	16#8008 => error state machine 
	16#8009 => timeout while waiting for data from server 
------------------------------------------------------------*)
VAR_IN_OUT
	xStartSend							: BOOL;
	aReceiveBuffer						: ARRAY [0..MAX_RECEIVE_TCP_CLIENT] OF BYTE;
	diReceiveCount						: DINT;
END_VAR
VAR
	m_State								: BYTE := 0;
	m_ReceiveBuffer						: ARRAY [0..MAX_RECEIVE_TCP_CLIENT_SOCKET] OF BYTE;
	m_Socket							: DINT;
	m_AddressInfo						: SOCKADDRESS;
	m_BytesReceived						: DINT;
	m_diReturn							: DINT;
	m_xReturn							: BOOL;
	m_IoCtlParameter  					: DINT := 1; (* IOCTL-Parameter for non-blocking mode of sockets *)
	i									: INT;
	T_Connect							: TON;
	m_count								: DINT;
	diOption							: DINT := 1;
	m_Blocking   						: DINT := 0;
END_VAR
IF xOpenConnection THEN
	(* State maschine *)
	CASE  m_State OF

	(* -------------------------------------------------------------------------*)
	STATE_CREATE:
			(* create socket descriptor*)
			m_Socket := SysSockCreate(diAddressFamily	:= SOCKET_AF_INET,
													 diType		:= SOCKET_STREAM,
													 diProtocol := SOCKET_IPPROTO_TCP);
			IF m_Socket >= 0 THEN
			(*Set Push-Bit*)
				IF ADR(%MW0)=16#30000000  OR ADR(%MW0)=16#20000000 THEN (*841 or 881*)
					SysSockSetOption(
						diSocket:=m_Socket,
						diLevel:=6,
						diOption:=SOCKET_TCP_NODELAY,
						pOptionValue:=ADR(diOption),
						diOptionLength:=SIZEOF(diOption));
				ELSE
						;
				END_IF
				m_State := STATE_IOCTL; (* succesful *)
			ELSE
				diError := 16#8001;  (* no socket descriptor available *)
				m_State := STATE_ERROR_TRAP;
			END_IF

	(* -------------------------------------------------------------------------*)
	STATE_IOCTL: (* change  socket mode  to none blocking *)
		m_diReturn := SysSockIoctl( m_Socket, SOCKET_FIONBIO, ADR(m_IoCtlParameter));
		IF m_diReturn <> 0 THEN
			m_AddressInfo.sin_family := SOCKET_AF_INET;
			m_AddressInfo.sin_port := SysSockNtohs(wPortNumber);
			m_AddressInfo.sin_addr := dwInetAddr;
			m_State := STATE_CONNECT;
		ELSE
			diError := 16#8004;  (* switching to none blocking mode fails *)
			m_State := STATE_ERROR_TRAP;
		END_IF


	(* -------------------------------------------------------------------------*)
	STATE_CONNECT: (* connect with server *)
		T_Connect(IN:=TRUE , PT:=tConnectWatchdogTime);(*activate watchdog for establishing connection to a server*)
		m_xReturn := SysSockConnect ( m_Socket, ADR(m_AddressInfo),  SIZEOF(m_AddressInfo));
		IF m_xReturn THEN (* succesful *)
			IF xStartSend THEN
				m_State := STATE_TX;(*transmit data*)
			ELSE
				m_State := STATE_RX;(*wait for data from server*)
			END_IF
			xConnected:=TRUE;
			T_Connect(IN:=FALSE);
		ELSE
			IF T_Connect.Q THEN
				diError := 16#8006;  (* connect fails *)
				xConnected:=FALSE;
				T_Connect(IN:=FALSE);
				m_State := STATE_ERROR_TRAP;
				SysSockClose( m_Socket);
			ELSE
				m_State := STATE_CONNECT;(*client still  tries to set up connection*)
			END_IF
		END_IF


	STATE_TX:	 (* send TCP-message *)
		m_diReturn := SysSockSend(diSocket := m_Socket,
								  pbyBuffer := ADR(ptSendData^[0]),
								  diBufferSize := diSendCount-m_count,
								  diFlags := 0);

		CASE m_diReturn OF
		-1:	(* ERROR *)
			T_Connect(IN:=TRUE , PT:=CONNECT_WATCHDOG_TIME);(*activate watchdog to check communication*)
			IF t_Connect.Q THEN
				diError := 16#8007;
				T_Connect(IN:=FALSE);
				m_State:=STATE_CLOSE;
			END_IF
		0: (* socket was "gracefully closed" *)
			m_State := STATE_CLOSE;
			diError := 16#8003;
		ELSE (* succesful *)
			m_count:=m_count+m_diReturn;
			IF m_count>=diSendCount THEN
				diError := 16#0000;
				m_State := STATE_RX;
				m_count:=0;
				xStartSend:=FALSE;
			END_IF
			T_Connect(IN:=FALSE);
		END_CASE

	(* -------------------------------------------------------------------------*)
	STATE_RX: (* process receive data *)
			m_BytesReceived := SysSockRecv(	diSocket 	:= m_Socket,
										pbyBuffer 	:= ADR(m_ReceiveBuffer),		(* Address of receive buffer *)
										diBufferSize:= SIZEOF(m_ReceiveBuffer),
										diFlags		:= 0);

			CASE m_BytesReceived OF
			-1:	(* No data available or error occured *)
				T_Connect(IN:=TRUE , PT:=tConnectWatchdogTime);(*activate watchdog to check communication*)
				IF t_Connect.Q THEN
					diError:=16#8009;
					T_Connect(IN:=FALSE);
					m_State:=STATE_CLOSE;
				END_IF
				IF xStartSend THEN
					m_State:=STATE_TX	;(* WAIT IN THIS STATE  and check for arriving data or new send command*)
				END_IF;
			0: (* socket was "gracefully closed"  *)
				m_State:=STATE_CLOSE;
				diError := 16#8003;
			ELSE (* succesful *)
				diError := 16#0000;
				T_Connect(IN:=FALSE);
				(* Copy received data into receive buffer *)
				FOR i:= 0 TO DINT_TO_INT(m_BytesReceived	)-1 DO
					aReceiveBuffer[diReceiveCount]:= m_ReceiveBuffer[i];
					diReceiveCount:=(diReceiveCount+1) MOD SIZEOF(aReceiveBuffer);
				END_FOR

			END_CASE

	(* -------------------------------------------------------------------------*)
	STATE_CLOSE : (* close socket *)
		IF ADR(%MW0)=16#30000000  OR ADR(%MW0)=16#20000000 THEN (*841 or 881*)
			;
		ELSE
			SysSockShutdown(m_Socket, 0);;(*870*)
		END_IF
		m_xReturn := SysSockClose( m_Socket);
		m_Socket := -1;
		m_State := 0; (* succesful *)
		xConnected:=FALSE;
		T_Connect(IN:=FALSE);
	(* -------------------------------------------------------------------------*)
	STATE_ERROR_TRAP: (* error handling *)
		xConnected:=FALSE;

	ELSE  (* Bad FSM code trap  *)
			m_State:= STATE_ERROR_TRAP;
			diError:= 16#8008;
	END_CASE

ELSE(*close connection*)
	IF m_Socket >= 0 THEN
		IF ADR(%MW0)=16#30000000  OR ADR(%MW0)=16#20000000 THEN (*841 or 881*)
			;
		ELSE
			SysSockShutdown(m_Socket, 0);;(*870*)
		END_IF
		SysSockClose( m_Socket);
	END_IF
	m_Socket := -1;
	diError := 16#0000;
	m_State := STATE_CREATE;
	xConnected:=FALSE;
	T_Connect(IN:=FALSE);
END_IF
END_FUNCTION_BLOCK

(* POU Utils Functions/DWORDSWAP, ST *)
FUNCTION DWORDSWAP:BOOL
VAR_INPUT
	pIn:POINTER TO ARRAY[1..4] OF BYTE;
	pOut:POINTER TO ARRAY[1..4] OF BYTE;
END_VAR
VAR
END_VAR
pOut^[1]:=pIn^[4];
pOut^[2]:=pIn^[3];
pOut^[3]:=pIn^[2];
pOut^[4]:=pIn^[1];
END_FUNCTION

(* POU Utils Functions/CHKSTRING, ST *)
FUNCTION CHKSTRING : BOOL
VAR_INPUT
	pString: POINTER TO BYTE;
	pPattern: POINTER TO BYTE;
END_VAR
VAR
END_VAR
CHKSTRING:=TRUE;
WHILE pPattern^<>0 AND CHKSTRING DO
	IF pPattern^<>pString^ THEN CHKSTRING:=FALSE; END_IF
	pString:=pString+1;
	pPattern:=pPattern+1;
END_WHILE
END_FUNCTION

(* POU TCP_Remote/Remote_Proc, ST *)
PROGRAM Remote_Proc
VAR
	s1:         	TCPSERVER;
	Enable: 		BOOL;
	Connected: 		BOOL;
	Error: 			DINT;

	TxData:			ARRAY[0..MAX_SEND_TCP_SERVER] OF BYTE;
	TxLen:			DINT;
	TxTrig:			BOOL;

	RxData:			ARRAY [0..MAX_RECEIVE_TCP_SERVER] OF BYTE;
	RxLen:			DINT;

	Status:			DINT;

	(* Command interpreter *)

	Cmd_Buf:		ARRAY [0..MAX_RECEIVE_TCP_SERVER] OF BYTE;
	Cmd_Buf_U16:	POINTER TO WORD;
	Cmd_Buf_INT:	POINTER TO INT;
	Cmd_BufLen:		WORD;
	Cmd_St:			WORD;

	Cmd_Obj:		WORD;
	Cmd_ObjIdx:		WORD;
	Cmd_C:			WORD;
	Cmd_R:			WORD;
	Cmd_CLen:		WORD;
	Cmd_RLen:		WORD;

	i : WORD;
	j : INT;


		(* per aggiornare la data e l'ora *)
	SetAnno: INT;
	SetMese: INT;
	SetGiorno: INT;
	SetOra: INT;
	SetMinuti: INT;
	SetSecondi: INT;


END_VAR
(*=== State machine ===*)
CASE Status OF
	0: (* Startup *)
		TxLen:=0; TxTrig:=FALSE;
		RxLen:=0;
		Enable:=TRUE;
		Status:=1;

	1: (* Wait incoming connection *)
		IF Connected THEN
			(* Log access *)
			LogEv(EL_Log,EO_VPN,1,5,'Remote');
			(* Send welcome message *)
			(*ADDSTRING(pTxData:=ADR(TxData), pString:=ADR(Remote_WELCOME), TxLen:=TxLen);
			TxTrig:=TRUE;*)
			Cmd_BufLen:=0;
			Cmd_St:=0;
			Status:=2;
		END_IF
		IF Error>1 THEN
			Enable:=FALSE;
			Status:=0;
		END_IF

	2: (* Wait command *)
		IF RxLen>0 THEN
			(*=== Interpreter start ===*)
			IF Cmd_BufLen+(RxLen/2)>=MAX_RECEIVE_TCP_SERVER THEN
				(* ERROR *)
				Cmd_BufLen:=0;
			ELSE
				i:=HEXTORAW(pString:=ADR(RxData), StringLen:=DINT_TO_WORD(RxLen), pData:=ADR(Cmd_Buf[Cmd_BufLen]));
				Cmd_BufLen:=Cmd_BufLen+i;
			END_IF
			IF Cmd_BufLen>=8 THEN
				Cmd_Buf_U16:=ADR(Cmd_Buf[6]);
				IF Cmd_BufLen>=(8+Cmd_Buf_U16^) THEN
					Cmd_CLen:=Cmd_Buf_U16^;
					Cmd_Buf_U16:=ADR(Cmd_Buf[0]); Cmd_Obj:=Cmd_Buf_U16^;
					Cmd_Buf_U16:=ADR(Cmd_Buf[2]); Cmd_ObjIdx:=Cmd_Buf_U16^;
					Cmd_Buf_U16:=ADR(Cmd_Buf[4]); Cmd_C:=Cmd_Buf_U16^;
					Command();
					Cmd_BufLen:=0;
				END_IF
			END_IF
			(*=== Interpreter end ===*)
			RxLen:=0;
		END_IF
		IF NOT Connected THEN
			Status:=0;
		END_IF

ELSE
	Status:=0;
END_CASE


(*=== Execute server lib ===*)
s1(
	xEnable				:= Enable,
	wPortNumber			:= Remote_PORT,
	tServerTimeOut		:= t#15m,
	ptSendData			:= ADR(TxData),
	diSendCount			:= TxLen,
	xStartSend			:= TxTrig,
	aReceiveBuffer		:= RxData,
	diReceiveCount		:= RxLen,
	xClientConnected	=> Connected,
	diError				=> Error
);
END_PROGRAM
ACTION Cmd_COMPINGRML:
(* Check index *)
IF Cmd_ObjIdx<>2 AND  Cmd_ObjIdx<>3  AND Cmd_ObjIdx<>4 THEN
	Cmd_R:=2;
	RETURN;
END_IF

(* Process command *)

CASE Cmd_C OF

	1:	(* Force UTA On *)
		CASE Cmd_ObjIdx OF

			2:	COMPRESSORE02.RELEASE_REQ := FALSE;
				COMPRESSORE02.RUN_REQ := TRUE;
				COMPRESSORE02.STOP_REQ 	:= FALSE;
				COMPRESSORE02.AgggiornoStartStop := TRUE;
			3:	COMPRESSORE03.RELEASE_REQ := FALSE;
				COMPRESSORE03.RUN_REQ := TRUE;
				COMPRESSORE03.STOP_REQ 	:= FALSE;
				COMPRESSORE03.AgggiornoStartStop := TRUE;
			4:	COMPRESSORE04.RELEASE_REQ := FALSE;
				COMPRESSORE04.RUN_REQ := TRUE;
				COMPRESSORE04.STOP_REQ 	:= FALSE;
				COMPRESSORE04.AgggiornoStartStop := TRUE;
		END_CASE

	2:	(* Force UTA Off *)
		CASE Cmd_ObjIdx OF

			2:	COMPRESSORE02.RELEASE_REQ := FALSE;
				COMPRESSORE02.STOP_REQ := TRUE;
				COMPRESSORE02.RUN_REQ	:= FALSE;
				COMPRESSORE02.AgggiornoStartStop := TRUE;
			3:	COMPRESSORE03.RELEASE_REQ := FALSE;
				COMPRESSORE03.STOP_REQ := TRUE;
				COMPRESSORE03.RUN_REQ	:= FALSE;
				COMPRESSORE03.AgggiornoStartStop := TRUE;
			4:	COMPRESSORE04.RELEASE_REQ := FALSE;
				COMPRESSORE04.STOP_REQ := TRUE;
				COMPRESSORE04.RUN_REQ	:= FALSE;
				COMPRESSORE04.AgggiornoStartStop := TRUE;
		END_CASE

	3:	(* Release force *)
		CASE Cmd_ObjIdx OF

			2:	COMPRESSORE02.RELEASE_REQ := TRUE;
				COMPRESSORE02.STOP_REQ := FALSE;
				COMPRESSORE02.RUN_REQ	:= FALSE;
				COMPRESSORE02.AgggiornoStartStop := TRUE;
			3:	COMPRESSORE03.RELEASE_REQ := TRUE;
				COMPRESSORE03.STOP_REQ := FALSE;
				COMPRESSORE03.RUN_REQ	:= FALSE;
				COMPRESSORE03.AgggiornoStartStop := TRUE;
			4:	COMPRESSORE04.RELEASE_REQ := TRUE;
				COMPRESSORE04.STOP_REQ := FALSE;
				COMPRESSORE04.RUN_REQ	:= FALSE;
				COMPRESSORE04.AgggiornoStartStop := TRUE;
		END_CASE

	4:	(* Release force *)
		CASE Cmd_ObjIdx OF

			2:	COMPRESSORE02.Carico_req := TRUE;
				COMPRESSORE02.AgggiornoStartStop := TRUE;
			3:	COMPRESSORE03.Carico_req := FALSE;
				COMPRESSORE03.AgggiornoStartStop := TRUE;
			4:	COMPRESSORE04.Carico_req := FALSE;
				COMPRESSORE04.AgggiornoStartStop := TRUE;
		END_CASE




	5: (* SET Comandi  *)
		CASE Cmd_ObjIdx OF
			2:	Cmd_Buf_U16:=ADR(Cmd_Buf[8]);
				COMPRESSORE02.ScriviCoil := DWORD_TO_BOOL(Cmd_Buf_U16^); 	(* 0 write on register - 1 write on coil *)
				Cmd_Buf_U16:=ADR(Cmd_Buf[10]);
				COMPRESSORE02.IndirizzoDaScrivere :=(Cmd_Buf_U16^); 				(* Address of the register / coil.  *)
				Cmd_Buf_U16:=ADR(Cmd_Buf[12]);
				COMPRESSORE02.DatoDaScrivere := (Cmd_Buf_U16^); 					(* The value to be written.  *)

			COMPRESSORE02.AgggiornoStartStop := TRUE;
				COMPRESSORE02.Refresh_Now := TRUE;

			3:	Cmd_Buf_U16:=ADR(Cmd_Buf[8]);
				COMPRESSORE03.ScriviCoil := DWORD_TO_BOOL(Cmd_Buf_U16^); 	(* 0 write on register - 1 write on coil *)
				Cmd_Buf_U16:=ADR(Cmd_Buf[10]);
				COMPRESSORE03.IndirizzoDaScrivere :=(Cmd_Buf_U16^); 				(* Address of the register / coil.  *)
				Cmd_Buf_U16:=ADR(Cmd_Buf[12]);
				COMPRESSORE03.DatoDaScrivere := (Cmd_Buf_U16^); 					(* The value to be written.  *)

			COMPRESSORE03.AgggiornoStartStop := TRUE;
				COMPRESSORE03.Refresh_Now := TRUE;

			4:	Cmd_Buf_U16:=ADR(Cmd_Buf[8]);
				COMPRESSORE04.ScriviCoil := DWORD_TO_BOOL(Cmd_Buf_U16^); 	(* 0 write on register - 1 write on coil *)
				Cmd_Buf_U16:=ADR(Cmd_Buf[10]);
				COMPRESSORE04.IndirizzoDaScrivere :=(Cmd_Buf_U16^); 				(* Address of the register / coil.  *)
				Cmd_Buf_U16:=ADR(Cmd_Buf[12]);
				COMPRESSORE04.DatoDaScrivere := (Cmd_Buf_U16^); 					(* The value to be written.  *)

			COMPRESSORE04.AgggiornoStartStop := TRUE;
				COMPRESSORE04.Refresh_Now := TRUE;
		END_CASE




ELSE
	Cmd_R:=3;
END_CASE
END_ACTION
ACTION Cmd_COMPINGRR:
(* Check index *)
IF Cmd_ObjIdx<>1 AND  Cmd_ObjIdx<>5THEN
	Cmd_R:=2;
	RETURN;
END_IF

(* Process command *)

CASE Cmd_C OF

	1:	(* Force UTA On *)
		CASE Cmd_ObjIdx OF

			1:	COMPRESSORE01.RELEASE_REQ := FALSE;
				COMPRESSORE01.RUN_REQ := TRUE;
				COMPRESSORE01.STOP_REQ 	:= FALSE;
				COMPRESSORE01.AgggiornoStartStop := TRUE;
			5:	COMPRESSORE05.RELEASE_REQ := FALSE;
				COMPRESSORE05.RUN_REQ := TRUE;
				COMPRESSORE05.STOP_REQ 	:= FALSE;
				COMPRESSORE05.AgggiornoStartStop := TRUE;
		END_CASE

	2:	(* Force UTA Off *)
		CASE Cmd_ObjIdx OF

			1:	COMPRESSORE01.RELEASE_REQ := FALSE;
				COMPRESSORE01.STOP_REQ := TRUE;
				COMPRESSORE01.RUN_REQ	:= FALSE;
				COMPRESSORE01.AgggiornoStartStop := TRUE;
			5:	COMPRESSORE05.RELEASE_REQ := FALSE;
				COMPRESSORE05.STOP_REQ := TRUE;
				COMPRESSORE05.RUN_REQ	:= FALSE;
				COMPRESSORE05.AgggiornoStartStop := TRUE;
		END_CASE

	3:	(* Release force *)
		CASE Cmd_ObjIdx OF

			1:	COMPRESSORE01.RELEASE_REQ := TRUE;
				COMPRESSORE01.STOP_REQ := FALSE;
				COMPRESSORE01.RUN_REQ	:= FALSE;
				COMPRESSORE01.AgggiornoStartStop := TRUE;
			5:	COMPRESSORE05.RELEASE_REQ := TRUE;
				COMPRESSORE05.STOP_REQ := FALSE;
				COMPRESSORE05.RUN_REQ	:= FALSE;
				COMPRESSORE05.AgggiornoStartStop := TRUE;
		END_CASE
	4:	(* Release force *)
		CASE Cmd_ObjIdx OF

			1:	COMPRESSORE01.Carico_req := TRUE;
				COMPRESSORE01.AgggiornoStartStop := TRUE;
			5:	COMPRESSORE05.Carico_req := FALSE;
				COMPRESSORE05.AgggiornoStartStop := TRUE;

		END_CASE




	5: (* SET Comandi  *)
		CASE Cmd_ObjIdx OF
			1:	Cmd_Buf_U16:=ADR(Cmd_Buf[8]);
				COMPRESSORE01.ScriviCoil := DWORD_TO_BOOL(Cmd_Buf_U16^); 	(* 0 write on register - 1 write on coil *)
				Cmd_Buf_U16:=ADR(Cmd_Buf[10]);
				COMPRESSORE01.IndirizzoDaScrivere :=(Cmd_Buf_U16^); 				(* Address of the register / coil.  *)
				Cmd_Buf_U16:=ADR(Cmd_Buf[12]);
				COMPRESSORE01.DatoDaScrivere := (Cmd_Buf_U16^); 					(* The value to be written.  *)

				COMPRESSORE01.AgggiornoStartStop := TRUE;
				COMPRESSORE01.Refresh_Now := TRUE;

			5:	Cmd_Buf_U16:=ADR(Cmd_Buf[8]);
				COMPRESSORE05.ScriviCoil := DWORD_TO_BOOL(Cmd_Buf_U16^); 	(* 0 write on register - 1 write on coil *)
				Cmd_Buf_U16:=ADR(Cmd_Buf[10]);
				COMPRESSORE05.IndirizzoDaScrivere :=(Cmd_Buf_U16^); 				(* Address of the register / coil.  *)
				Cmd_Buf_U16:=ADR(Cmd_Buf[12]);
				COMPRESSORE05.DatoDaScrivere := (Cmd_Buf_U16^); 					(* The value to be written.  *)

				COMPRESSORE05.AgggiornoStartStop := TRUE;
				COMPRESSORE05.Refresh_Now := TRUE;
		END_CASE




ELSE
	Cmd_R:=3;
END_CASE
END_ACTION
ACTION Cmd_SYS:
(* Check index *)
IF Cmd_ObjIdx<>0 THEN
	Cmd_R:=2;
	RETURN;
END_IF

(* Process command *)
CASE Cmd_C OF

	0: (* ECHO *)
		IF Cmd_CLen<>0 THEN
			TxLen:=0;
		END_IF

	1: (* LOG REQUEST *)
		(*LogTrig(); *)
		PLC_PRG.RichiestaDaRemoto:=TRUE;


	2: (* REARM *)
		Sys.Warning:=FALSE;
		Sys.Alarm:=FALSE;
		Sys.AlarmStop:=FALSE;

	3: (* GET INFO1 *)
		Cmd_RLen:=6;
		TxLen:=TxLen+RAWTOHEX(ADR(Plant_SN),4,ADR(TxData[TxLen]));
		TxLen:=TxLen+RAWTOHEX(ADR(Plant_SW_VER),2,ADR(TxData[TxLen]));


	4: (*  Scrivo i Parametri gestione Impianto   *)

			Cmd_Buf_U16:=ADR(Cmd_Buf[8]);
			DelayAllarmeTemperaturaNonRaggiunta := Cmd_Buf_U16^; 			(* Ritardo Allarme dall'avvio Caldaia*)
			Cmd_Buf_U16:=ADR(Cmd_Buf[10]);
			DeltaInterventoAllarmeTempeaturaNonRaggiuta := Cmd_Buf_U16^;	(* Delta Soglia Temperatura per Allarme Temperatura Non Raggiunta *)
			Cmd_Buf_U16:=ADR(Cmd_Buf[12]);
			OffsetSetPointManuale := Cmd_Buf_U16^; 							(* Offest Perdite Scambiatore 1  *)
			Cmd_Buf_U16:=ADR(Cmd_Buf[14]);
			OffsetSetPointManuale2 := Cmd_Buf_U16^; 						(* Offest Perdite Scambiatore 1  *)
			Cmd_Buf_U16:=ADR(Cmd_Buf[12]);
			BitAbilitaBoost :=INT_TO_BOOL( Cmd_Buf_U16^); 					(* Abilitazione controllo Boost  *)
			Cmd_Buf_U16:=ADR(Cmd_Buf[14]);
			RifOffsetBoost := Cmd_Buf_U16^; 								(* Offset al Setpoint della Caldaia per azione di Boost  *)


	5: (*  Leggi i parametri gestione Impianto  *)

			Cmd_RLen:=18;
			j:=(DelayAllarmeTemperaturaNonRaggiunta);   				(* Ritardo Allarme dall'avvio Caldaia*)
			TxLen:=TxLen+RAWTOHEX(ADR(j),2,ADR(TxData[TxLen]));
			j:=(DeltaInterventoAllarmeTempeaturaNonRaggiuta);			(* Delta Soglia Temperatura per Allarme Temperatura Non Raggiunta *)
			TxLen:=TxLen+RAWTOHEX(ADR(j),2,ADR(TxData[TxLen]));
			j:=(OffsetSetPointManuale);									(* Offest Perdite Scambiatore 1  *)
			TxLen:=TxLen+RAWTOHEX(ADR(j),2,ADR(TxData[TxLen]));
			j:=(OffsetSetPointManuale2);								(* Offest Perdite Scambiatore 2  *)
			TxLen:=TxLen+RAWTOHEX(ADR(j),2,ADR(TxData[TxLen]));
			j:=BOOL_TO_INT(BitAbilitaBoost);							(* Abilitazione controllo Boost  *)
			TxLen:=TxLen+RAWTOHEX(ADR(j),2,ADR(TxData[TxLen]));
			j:=BOOL_TO_INT(BitAbilitaBoost);										(* Offset al Setpoint della Caldaia per azione di Boost   *)
			TxLen:=TxLen+RAWTOHEX(ADR(j),2,ADR(TxData[TxLen]));




	6: (*  Scrivo i Parametri gestione Impianto - Antigelo   *)

			Cmd_Buf_U16:=ADR(Cmd_Buf[8]);
			SogliaMinStartAntigelo := Cmd_Buf_U16^; 			(* Soglia mininma Start Antigelo *)
			Cmd_Buf_U16:=ADR(Cmd_Buf[10]);
			SogliaMinStopAntigelo := Cmd_Buf_U16^;				(* Soglia Massima Stop Antigelo *)
			Cmd_Buf_U16:=ADR(Cmd_Buf[12]);
			BitAbilitaAntigelo :=INT_TO_BOOL( Cmd_Buf_U16^); 	(* Abilitazione Antigelo  *)

	7: (*  Leggi i parametri gestione Impianto - Antigelo *)

			Cmd_RLen:=14;
			j:=(SogliaMinStartAntigelo); 							(* Soglia mininma Start Antigelo *)
			TxLen:=TxLen+RAWTOHEX(ADR(j),2,ADR(TxData[TxLen]));
			j:=(SogliaMinStopAntigelo);								(* Soglia Massima Stop Antigelo *)
			TxLen:=TxLen+RAWTOHEX(ADR(j),2,ADR(TxData[TxLen]));
			j:=BOOL_TO_INT(BitAbilitaAntigelo);						(* Abilitazione Antigelo  *)
			TxLen:=TxLen+RAWTOHEX(ADR(j),2,ADR(TxData[TxLen]));

(*	10: (*  Scrivo i Parametri per la gestione della velocità dei circolatori sui primari   *)

			Cmd_Buf_U16:=ADR(Cmd_Buf[8]);
			PercVelMin := Cmd_Buf_U16^;
			Cmd_Buf_U16:=ADR(Cmd_Buf[10]);
			PercVelMax := Cmd_Buf_U16^;
			Cmd_Buf_U16:=ADR(Cmd_Buf[12]);
			ErroreTempMax := Cmd_Buf_U16^;
			Cmd_Buf_U16:=ADR(Cmd_Buf[14]);
			ErroreTempMin := Cmd_Buf_U16^;

	11: (*  Leggo i Parametri per la gestione della velocità dei circolatori sui primari   *)

			Cmd_RLen:=8;
			j:=(PercVelMin);
			TxLen:=TxLen+RAWTOHEX(ADR(j),2,ADR(TxData[TxLen]));
			j:=(PercVelMax);
			TxLen:=TxLen+RAWTOHEX(ADR(j),2,ADR(TxData[TxLen]));
			j:=(ErroreTempMax);
			TxLen:=TxLen+RAWTOHEX(ADR(j),2,ADR(TxData[TxLen]));
			j:=(ErroreTempMin);
			TxLen:=TxLen+RAWTOHEX(ADR(j),2,ADR(TxData[TxLen]));


	12: (*  Scrivo i Parametri per la gestione della velocità dei circolatori sui primari   *)


				Cmd_Buf_U16:=ADR(Cmd_Buf[8]);
				CAS01.DeltaTempThr := Cmd_Buf_U16^;
				Cmd_Buf_U16:=ADR(Cmd_Buf[10]);
				CAS01.Tmonitor_Off := DWORD_TO_TIME((Cmd_Buf_U16^)*60*1000);
				Cmd_Buf_U16:=ADR(Cmd_Buf[12]);
				CAS01.Tmonitor_On := DWORD_TO_TIME((Cmd_Buf_U16^)*60*1000);

	13: (*  Leggo i Parametri per la gestione della velocità dei circolatori sui primari   *)


				Cmd_RLen:=6;
				j:=(CAS01.DeltaTempThr);
				TxLen:=TxLen+RAWTOHEX(ADR(j),2,ADR(TxData[TxLen]));
				j:=DWORD_TO_WORD(TIME_TO_DWORD((CAS01.Tmonitor_Off)/60/1000));
				TxLen:=TxLen+RAWTOHEX(ADR(j),2,ADR(TxData[TxLen]));
				j:=DWORD_TO_WORD(TIME_TO_DWORD((CAS01.Tmonitor_On)/60/1000));
				TxLen:=TxLen+RAWTOHEX(ADR(j),2,ADR(TxData[TxLen]));


*)


	14: (*  Imposto data e ora del PLC  *)


			Cmd_Buf_U16:=ADR(Cmd_Buf[8]);
			SetAnno:= Cmd_Buf_U16^; 												(* Anno *)
			Cmd_Buf_U16:=ADR(Cmd_Buf[10]);
			SetMese:= Cmd_Buf_U16^;												 	(* mese *)
			Cmd_Buf_U16:=ADR(Cmd_Buf[12]);
			SetGiorno:=( Cmd_Buf_U16^);											 	(* Giorno *)
			Cmd_Buf_U16:=ADR(Cmd_Buf[14]);
			SetOra:=( Cmd_Buf_U16^); 												(* ora *)
			Cmd_Buf_U16:=ADR(Cmd_Buf[16]);
			SetMinuti:= ( Cmd_Buf_U16^);										 	(* Minuti *)
			Cmd_Buf_U16:=ADR(Cmd_Buf[18]);
			SetSecondi:= ( Cmd_Buf_U16^);										 	(* secondi *)

	(*		SysRtcSetTime(SetDataTime(DWORD_TO_INT(ADR(Cmd_Buf[8])),				(* Anno *)
										DWORD_TO_INT(ADR(Cmd_Buf[10])),				(* mese *)
										DWORD_TO_INT(ADR(Cmd_Buf[11])),				(* Giorno *)
										DWORD_TO_INT(ADR(Cmd_Buf[12])),				(* ora *)
										DWORD_TO_INT(ADR(Cmd_Buf[13])),				(* Minuti *)
										DWORD_TO_INT(ADR(Cmd_Buf[14]))				(* secondi *)
										)); *)

		SysRtcSetTime((SetDataTime(SetAnno,SetMese,SetGiorno,SetOra,SetMinuti,SetSecondi)));


ELSE
	Cmd_R:=3;
END_CASE
END_ACTION
ACTION Command:
(* Default response OK/NODATA *)
Cmd_R:=0;
Cmd_RLen:=0;
TxLen:=16;

(* Check object *)
CASE Cmd_Obj OF

	EO_SYS:
		Cmd_SYS();

	EO_COMPINGRR:
		Cmd_COMPINGRR();

	EO_COMPINGRML:
		Cmd_COMPINGRML();

ELSE
	Cmd_R:=1;
END_CASE

(* Generate response *)
IF TxLen>0 THEN
	RAWTOHEX(ADR(Cmd_Obj)	,2,ADR(TxData[ 0]));
	RAWTOHEX(ADR(Cmd_ObjIdx),2,ADR(TxData[ 4]));
	RAWTOHEX(ADR(Cmd_R)		,2,ADR(TxData[ 8]));
	RAWTOHEX(ADR(Cmd_RLen)	,2,ADR(TxData[12]));
	TxTrig:=TRUE;
END_IF
END_ACTION

(* POU Utils Functions/TCPSERVER, ST *)
FUNCTION_BLOCK TCPSERVER
(***********************************************************************************************************	*)
(* Version: 1.6                                    			          											*)
(* Date: 11.02.2011                                   					          							    *)
(***********************************************************************************************************	*)
(* WAGO Kontakttechnik GmbH Hansastr. 27 32423 Minden(Westf.)													*)
(* Tel. +0049 571/887-0 Fax. +0049 571/887-0																	*)
(* Author: VB																									*)
(***********************************************************************************************************	*)
(*Description:	A TCP server to read and write data													       		*)
(*Historie:																										*)
(*Version 1.6: 11.02.2011: Changes according to 750-880/881											 			*)
(*Version 1.5: 27.11.2008 Bugfix allow reuse port																*)
(*Version 1.4: 13.10.2008 Bugfix transmitting large data														*)
(*Version 1.3: 15.01.2007 Changes according to FW11																*)
(*Version 1.2: 09.03.2006 Changes for socket handle 0											       			*)
(*Version 1.1: 14.02.2005 Release																				*)
(***********************************************************************************************************	*)
VAR CONSTANT
	STATE_INIT     				 : BYTE:= 0;
	STATE_OPEN     				 : BYTE:= 1;
	STATE_TX       				 : BYTE:= 20;
	STATE_RX       				 : BYTE:= 30;
	STATE_CLOSE    				 : BYTE:= 40;
	STATE_ERROR_TRAP		 	 : BYTE:= 200;
END_VAR
VAR_INPUT
	xEnable    					: BOOL;	 (* Set TRUE to enable function block *)
	wPortNumber					: WORD;  (* Port *)
	tServerTimeOut				: TIME:=t#50s;
	ptSendData					: POINTER TO ARRAY[0..MAX_SEND_TCP_SERVER] OF BYTE;
	diSendCount					: DINT;
END_VAR
VAR_OUTPUT
	xClientConnected  			: BOOL:= FALSE;
	diError 					: DINT:= 0;
END_VAR
(* Status Codes -----------------------------------------
	16#8001 => No socket descriptor available 
	16#8002 => SysSockBind fails 
	16#8003 => SysSockListen fails 
	16#8004 => switching to none blocking mode fails
	16#8005 => SysSockClose() returns FALSE 
    16#8006 => SysSockConnect() fails
    16#8007 => SysSockSend() fails
	16#8008 => error state machine 
	16#8009 => timeout while waiting for data from server 
	16#0001 => server waiting for client to establish connection
------------------------------------------------------------*)
VAR_IN_OUT
	xStartSend					: BOOL;
	aReceiveBuffer				: ARRAY [0..MAX_RECEIVE_TCP_SERVER] OF BYTE;
	diReceiveCount				: DINT;
END_VAR

VAR
	m_State    					: BYTE:= 0;
	m_ReceiveBuffer				: ARRAY [0..MAX_RECEIVE_TCP_SERVER_SOCKET] OF BYTE;
	m_ServerSocket				: DINT:= SOCKET_INVALID;
	m_Socket					: DINT:= SOCKET_INVALID;
	m_AddressInfo				: SOCKADDRESS;
	m_BytesReceived				: DINT;
	m_diReturn					: DINT;
	m_xReturn					: BOOL;
	m_SizeSockadr				: DWORD;
	m_ConnectionWatchdog		: TON;
	m_Flags						: DINT;
	m_NoneBlocking   			: DINT:= 1;
	m_Blocking   				: DINT:= 0;
	i							: INT;
	m_count						: DINT;
	diOption					: DINT := 1;
	on: DINT;
END_VAR
IF xEnable THEN
	CASE m_State OF
		STATE_INIT:
			(* Create Socket *)
			m_ServerSocket:= SysSockCreate( SOCKET_AF_INET, SOCKET_STREAM, 0);
			IF m_ServerSocket = SOCKET_INVALID THEN
				(* *)
				diError:= 16#8001;
				m_State:= STATE_ERROR_TRAP;
				RETURN;
			ELSE
				;
			END_IF
			(* Address bindings *)
			(********************)
			on:=1;
			SysSockSetOption( m_ServerSocket, SOCKET_SOL, SOCKET_SO_REUSEADDR, ADR(on), SIZEOF(on) );

			m_AddressInfo.sin_family:= SOCKET_AF_INET;
			m_AddressInfo.sin_port  := SysSockHtons( wPortNumber);
			m_AddressInfo.sin_addr  := SOCKET_INADDR_ANY;
			IF NOT SysSockBind( m_ServerSocket, ADR(m_AddressInfo), SIZEOF(m_AddressInfo)) THEN
				diError:= 16#8002;
				m_State:= STATE_ERROR_TRAP;
				RETURN;
			END_IF
			(* Wait for connections *)
			(************************)
			IF NOT SysSockListen( m_ServerSocket, 1) THEN
				diError:= 16#8003;
				m_State:= STATE_ERROR_TRAP;
			END_IF

			(* Puts SOCKET in NonBlocking mode *)
			m_diReturn:= SysSockIoctl( m_ServerSocket, SOCKET_FIONBIO, ADR(m_NoneBlocking));

			m_State:= STATE_OPEN;


		STATE_OPEN: 	(* Waiting for incomming connection *)
				m_SizeSockadr:=SIZEOF(m_AddressInfo);
				m_Socket:= SysSockAccept( m_ServerSocket, ADR(m_AddressInfo), ADR(m_SizeSockadr));
				diError:=State_open;
				IF m_Socket <> SOCKET_INVALID THEN
					xClientConnected:=TRUE;
					(*Set Push-Bit:new V1.5*)
					IF ADR(%MW0)=16#30000000  OR ADR(%MW0)=16#20000000 THEN (*841 or 881*)
						SysSockSetOption(
							diSocket:=m_Socket,
							diLevel:=6,
							diOption:=SOCKET_TCP_NODELAY,
							pOptionValue:=ADR(diOption),
							diOptionLength:=SIZEOF(diOption));
					ELSE
							;
					END_IF
					SysSockIoctl( m_Socket, SOCKET_FIONBIO, ADR(m_NoneBlocking));
					m_State:= STATE_RX;
					diError:=0;
				END_IF

		STATE_RX:
					m_BytesReceived:= SysSockRecv( m_Socket, ADR(m_ReceiveBuffer), SIZEOF(m_ReceiveBuffer), 0);
					CASE m_BytesReceived OF
					-1:(*no data available or error occured*)
						m_ConnectionWatchdog(IN:=TRUE , PT:=tServerTimeOut );
						IF m_connectionWatchdog.Q THEN
							m_State:= STATE_CLOSE;
							m_ConnectionWatchdog(IN:=FALSE);(*reset connection watchdog*)
							diError := 16#8009;
						END_IF
					0:(* socket was "gracefully closed"  *)
						m_State:= STATE_CLOSE;
						diError := 16#8003;
					ELSE
						(* Copy received data into receive buffer *)
						(********************************)
						FOR i:= 0 TO DINT_TO_INT(m_BytesReceived	)-1 DO
							aReceiveBuffer[diReceiveCount]:= m_ReceiveBuffer[i];
							diReceiveCount:=(diReceiveCount+1) MOD SIZEOF(aReceiveBuffer);
						END_FOR

						m_ConnectionWatchdog(IN:=FALSE);(*reset connection watchdog*)
					END_CASE

				(*send data*)
				IF xStartSend	 THEN
					m_State := STATE_TX;
				END_IF

	STATE_TX:	 (* send TCP-message *)
		m_diReturn := SysSockSend(diSocket := m_Socket,
								  pbyBuffer := ADR(ptSendData^[m_count]),(*geändert V1.4 bisher: [0] *)
								  diBufferSize := diSendCount-m_count,
								  diFlags :=m_Flags);
		CASE m_diReturn OF
		-1:	(* ERROR or data could not yet be send (V1.3 due to new FW11) *)
			m_ConnectionWatchdog(IN:=TRUE , PT:=tServerTimeOut );
			IF m_connectionWatchdog.Q THEN
				m_State:= STATE_CLOSE;
				m_ConnectionWatchdog(IN:=FALSE);(*reset connection watchdog*)
				diError := 16#8007;
			END_IF
		0: (* socket was "gracefully closed"  *)
			m_State := STATE_CLOSE;
			diError := 16#8003;
		ELSE (* succesful *)
			m_count:=m_count+m_diReturn;
			IF m_count>=diSendCount THEN
				diError := 16#0000;
				m_State := STATE_RX;
				m_count:=0;
				xStartSend:=FALSE;
			END_IF
			m_ConnectionWatchdog(IN:=FALSE);(*reset connection watchdog*)
		END_CASE


		STATE_CLOSE:	(* Close the server *)

		IF ADR(%MW0)=16#30000000  OR ADR(%MW0)=16#20000000 THEN (*841 or 881*)
			;
		ELSE
			IF m_Socket>=0 THEN
				SysSockShutdown(m_Socket, 0);;(*870*)
			END_IF
		END_IF
		IF m_Socket>=0 THEN
			SysSockClose( m_Socket);
		END_IF
		xClientConnected:= FALSE;
		m_State:= STATE_OPEN; (* Try to open the server again *)
		m_ConnectionWatchdog(IN:=FALSE);(*reset connection watchdog*)

		STATE_ERROR_TRAP: (* Error Read/Write socket  *)
			m_State:= STATE_ERROR_TRAP;

	ELSE  (* Bad FSM code trap  *)
			m_State:= STATE_ERROR_TRAP;
			diError:= 16#8008;
	END_CASE;
ELSE
	IF m_State <> STATE_INIT THEN
		IF ADR(%MW0)=16#30000000  OR ADR(%MW0)=16#20000000 THEN (*841 or 881*)
			;
		ELSE
			IF m_Socket>=0 THEN
				SysSockShutdown(m_Socket, 0);;(*870*)
			END_IF
		END_IF
		IF m_Socket>=0 THEN
			SysSockClose( m_Socket);
		END_IF
		IF ADR(%MW0)=16#30000000  OR ADR(%MW0)=16#20000000 THEN (*841 or 881*)
			;
		ELSE
			IF m_ServerSocket>=0 THEN
				SysSockShutdown(m_ServerSocket, 0);;(*870*)
			END_IF
		END_IF
		IF m_ServerSocket>=0 THEN
			SysSockClose( m_ServerSocket);
		END_IF
		xClientConnected:= FALSE;
		diError:= 0;
		m_State:= STATE_init; (* Try to open the server again *)
		m_ConnectionWatchdog(IN:=FALSE);(*reset connection watchdog*)
	END_IF
END_IF
END_FUNCTION_BLOCK

(* POU Utils Functions/HEXTORAW, ST *)
FUNCTION HEXTORAW : WORD
VAR_INPUT
	pString		: POINTER TO BYTE;
	StringLen	: WORD;
	pData		: POINTER TO BYTE;
END_VAR
VAR
	xl: WORD;
	xi: WORD;
	xr: BYTE;
END_VAR
xl:=0;
xi:=0;

WHILE xi<StringLen DO

	IF pString^>=97 AND pString^<=102 THEN
		xr := pString^ - 87;
	ELSIF pString^>=65 AND pString^<=70 THEN
		xr := pString^ - 55;
	ELSIF pString^>=48 AND pString^<=57 THEN
		xr := pString^ - 48;
	ELSE
		xr := 16;
	END_IF

	IF xr<16 THEN
		IF (xi AND 1)=0 THEN
			pData^ := xr * 16;
		ELSE
			pData^ := pData^ + xr;
			pData := pData + 1;
			xl := xl + 1;
		END_IF
	END_IF

	xi := xi + 1;
	pString := pString + 1;

END_WHILE

HEXTORAW:=xl;
END_FUNCTION

(* POU TCP_Remote/LogTrig, ST *)
FUNCTION LogTrig : BOOL
VAR
	s1 : STRING(160);
	i  : BYTE;
	j  : WORD;
	BitTest: BOOL;
END_VAR
BitTest:=TRUE;

(*

(*---------------------------------------------------------------*)
	Logger_Head();
(*---------------------------------------------------------------*)

PX01.AddLogData();
PX02.AddLogData();
PX03.AddLogData();
PX04.AddLogData();
Logger_Send();


Logger_Head();

(*
FOR i:=1 TO Plant_ANZ_INEPRO DO
	ANZ_INEPRO[i].AddLogData();
END_FOR *)
ANZ_INEPRO[1].AddLogData();
ANZ_INEPRO[2].AddLogData();
Logger_Send();


Logger_Head();

ANZ_INEPRO[3].AddLogData();
ANZ_INEPRO[4].AddLogData();
Logger_Send();


Logger_Head();
ANZ_INEPRO[5].AddLogData();

Logger_Send();


Logger_Head();

	COMPRESSORE01.AddLogData(ModBus:=MODB02);
	COMPRESSORE05.AddLogData(ModBus:=MODB02);
Logger_Send();


Logger_Head();
	COMPRESSORE02.AddLogData(ModBus:=MODB03);
	COMPRESSORE03.AddLogData(ModBus:=MODB03);
	COMPRESSORE04.AddLogData(ModBus:=MODB03);
Logger_Send();


Logger_Head();

	FPT01.AddLogData(ModBus:=MODB05);
	FPT02.AddLogData();
	FPT03.AddLogData();
	FPT04.AddLogData();
	FPT05.AddLogData();
	FPT06.AddLogData();
	FPT07.AddLogData();
	FPT08.AddLogData();
	FPT09.AddLogData();
	FPT10.AddLogData();

(*	ESSICATORE01.AddLogData(ModBus:=MODB04); *)
(*	ESSICATORE02.AddLogData(ModBus:=MODB04); *)



(*---------------------------------------------------------------*)
	Logger_Send();
(*---------------------------------------------------------------*)
*)
END_FUNCTION

(* POU Utils Functions/RAWTOHEX, ST *)
FUNCTION RAWTOHEX : WORD
VAR_INPUT
	pData: POINTER TO BYTE;
	DataLen: WORD;
	pString: POINTER TO BYTE;
END_VAR
VAR
	xl: WORD;
END_VAR
xl:=0;

WHILE DataLen>0 DO

	pString^ := (pData^ / 16#10) + 48 + (((pData^ / 16#10)/10)*7);
	pString:=pString+1;
	pString^ := (pData^ AND 16#0F)  + 48 + (((pData^ AND 16#0F)/10)*7);
	pString:=pString+1;
	pData:=pData+1;
	DataLen:=DataLen-1;
	xl:=xl+2;

END_WHILE

(*pString^:=0;*)

RAWTOHEX:=xl;
END_FUNCTION

(* POU Utils Functions/GestioneDataTime_DaOscat/SetDataTime, ST *)
FUNCTION SetDataTime : DT
VAR_INPUT
	year : INT;
	month : INT;
	day : INT;
	hour : INT;
	minute : INT;
	second : INT;
END_VAR

VAR
	count : INT;
END_VAR
(* Creazione variabiletipo DT per creare Orario da dare al PLC *)


IF month > 2 THEN
	count := (month - 1) * 30;
	IF month > 7 THEN count := count + SHR(month - 3,1); ELSE count := count + SHR(month - 4,1); END_IF;
	(* chech for leap year and add one day if true *)
	IF SHL(year,14) = 0 THEN count := count + 1; END_IF;
ELSE
	count := (month - 1) * 31;
END_IF;


SetDataTime := DWORD_TO_DT(DATE_TO_DWORD( DWORD_TO_DATE((INT_TO_DWORD(count + day - 1) + SHR(INT_TO_DWORD(year) * 1461 - 2878169, 2)) * 86400))
				+ INT_TO_DWORD(SECOND)
				+ INT_TO_DWORD(MINUTE) * 60
				+ INT_TO_DWORD(HOUR) * 3600);
END_FUNCTION

(* POU Plant/SYS_Proc, ST *)
PROGRAM SYS_Proc
VAR
	fALARM_PB		:FLT_TAP;
	fALARM_TB		:FLT_TAP;
	fALARM_PM		:FLT_TAP;
	fALARM_ALARM_PM_PB_TB		:FLT_TAP;

(*	fGZB_ST			:FLT_TAP;  (* GATEWAY ZIGBEE *)*)
	fVPN_ST1		:FLT_TAP;  (* VPN CONNECT *)
	fVPN_ST2		:FLT_TAP;  (* VPN STATUS *)
	fKEY_CT_ST		:FLT_TAP;  (* DOOR1 *)
	fKEY_SCT_ST		:FLT_TAP;  (* DOOR2 *)
	fKEY_QE_ST		:FLT_TAP;  (* DOOR3 *)


	fBostAttivo	:FLT_TAP;

	fALARM_MancatoRaggiungimentoAcqua		:FLT_TAP;
	DelayfALARM_MancatoRaggiungimentoAcqua:TON;

END_VAR
(*************** ISPESL *****************)
(*
fALARM_PB(IN:=ALARM_PB);
IF fALARM_PB.EVH THEN
	LogEv(EL_AlarmStop,EO_PBV,1,1,'Over_Pressure_Alarm');
END_IF

fALARM_TB(IN:=ALARM_TB);
IF fALARM_TB.EVH THEN
	LogEv(EL_AlarmStop,EO_TBV,1,1,'Over_Temperature_Alarm');
END_IF

fALARM_PM(IN:=ALARM_PM);
IF fALARM_PM.EVH THEN
	LogEv(EL_AlarmStop,EO_PMV,1,1,'Under_Pressure_Alarm');
END_IF
*)
(*
fALARM_ALARM_PM_PB_TB(IN:=ALARM_PM_PB_TB);
IF fALARM_ALARM_PM_PB_TB.EVH THEN
	LogEv(EL_AlarmStop,EO_PMV,1,1,'Allarmi_ISPESL');
END_IF
*)





(****************************************)

